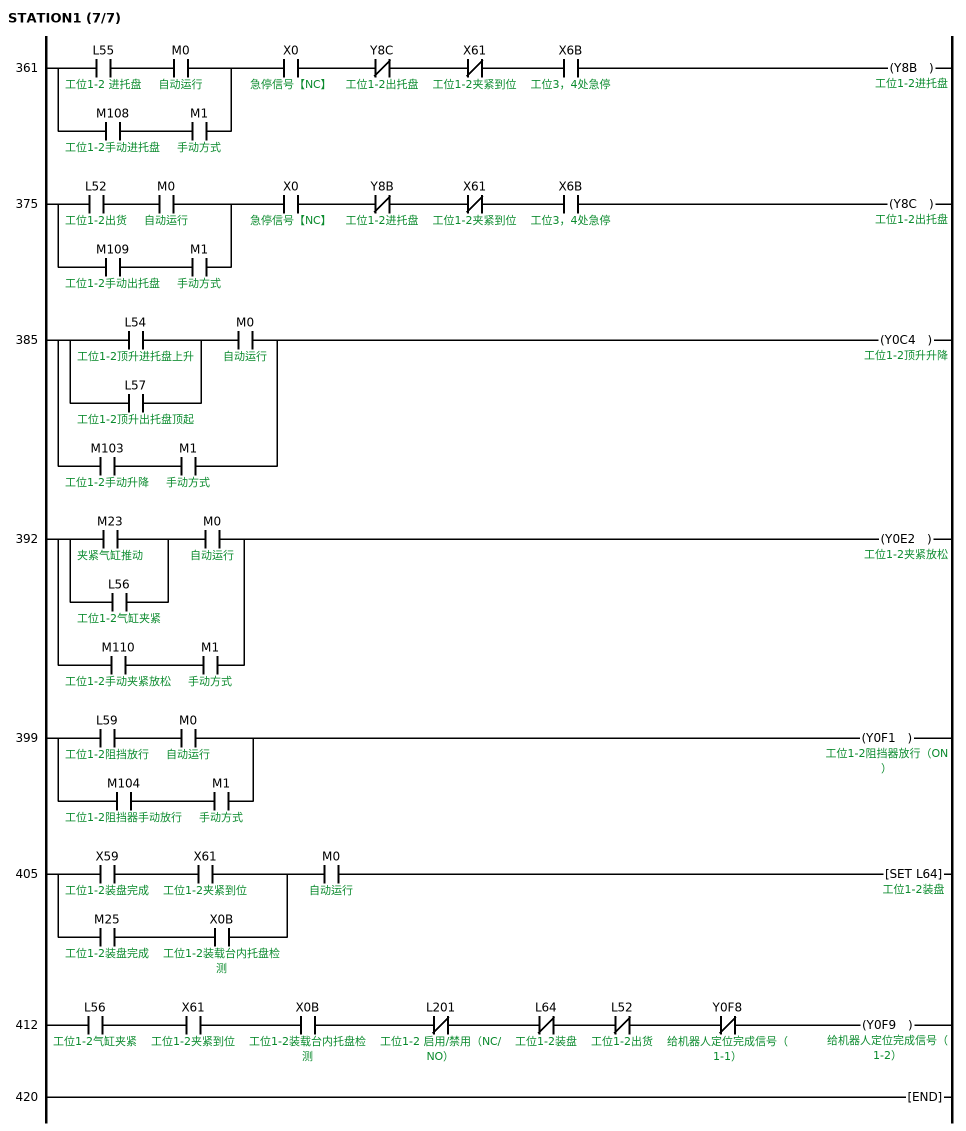
[picture p48: ladder of STATION1, rungs at steps 361 to 420]
361   LD      L55  ; 工位1-2 进托盘
      AND     M0  ; 自动运行
      LD      M108  ; 工位1-2手动进托盘
      AND     M1  ; 手动方式
      ORB
      AND     X0  ; 急停信号【NC】
      ANI     Y8C  ; 工位1-2出托盘
      ANI     X61  ; 工位1-2夹紧到位
      AND     X6B  ; 工位3，4处急停
      OUT     Y8B  ; 工位1-2进托盘
        [note] 1-2
375   LD      L52  ; 工位1-2出货
      AND     M0  ; 自动运行
      LD      M109  ; 工位1-2手动出托盘
      AND     M1  ; 手动方式
      ORB
      AND     X0  ; 急停信号【NC】
      ANI     Y8B  ; 工位1-2进托盘
      ANI     X61  ; 工位1-2夹紧到位
      AND     X6B  ; 工位3，4处急停
      OUT     Y8C  ; 工位1-2出托盘
385   LD      L54  ; 工位1-2顶升进托盘上升
      OR      L57  ; 工位1-2顶升出托盘顶起
      AND     M0  ; 自动运行
      LD      M103  ; 工位1-2手动升降
      AND     M1  ; 手动方式
      ORB
      OUT     Y0C4  ; 工位1-2顶升升降
392   LD      M23  ; 夹紧气缸推动
      OR      L56  ; 工位1-2气缸夹紧
      AND     M0  ; 自动运行
      LD      M110  ; 工位1-2手动夹紧放松
      AND     M1  ; 手动方式
      ORB
      OUT     Y0E2  ; 工位1-2夹紧放松
399   LD      L59  ; 工位1-2阻挡放行
      AND     M0  ; 自动运行
      LD      M104  ; 工位1-2阻挡器手动放行
      AND     M1  ; 手动方式
      ORB
      OUT     Y0F1  ; 工位1-2阻挡器放行（ON）
405   LD      X59  ; 工位1-2装盘完成
      AND     X61  ; 工位1-2夹紧到位
      LD      M25  ; 工位1-2装盘完成
      AND     X0B  ; 工位1-2装载台内托盘检测
      ORB
      AND     M0  ; 自动运行
      SET     L64  ; 工位1-2装盘
412   LD      L56  ; 工位1-2气缸夹紧
      AND     X61  ; 工位1-2夹紧到位
      AND     X0B  ; 工位1-2装载台内托盘检测
      ANI     L201  ; 工位1-2 启用/禁用（NC/NO）
      ANI     L64  ; 工位1-2装盘
      ANI     L52  ; 工位1-2出货
      ANI     Y0F8  ; 给机器人定位完成信号（1-1）
      OUT     Y0F9  ; 给机器人定位完成信号（1-2）
420   END
END_PROGRAM

PROGRAM STATION2
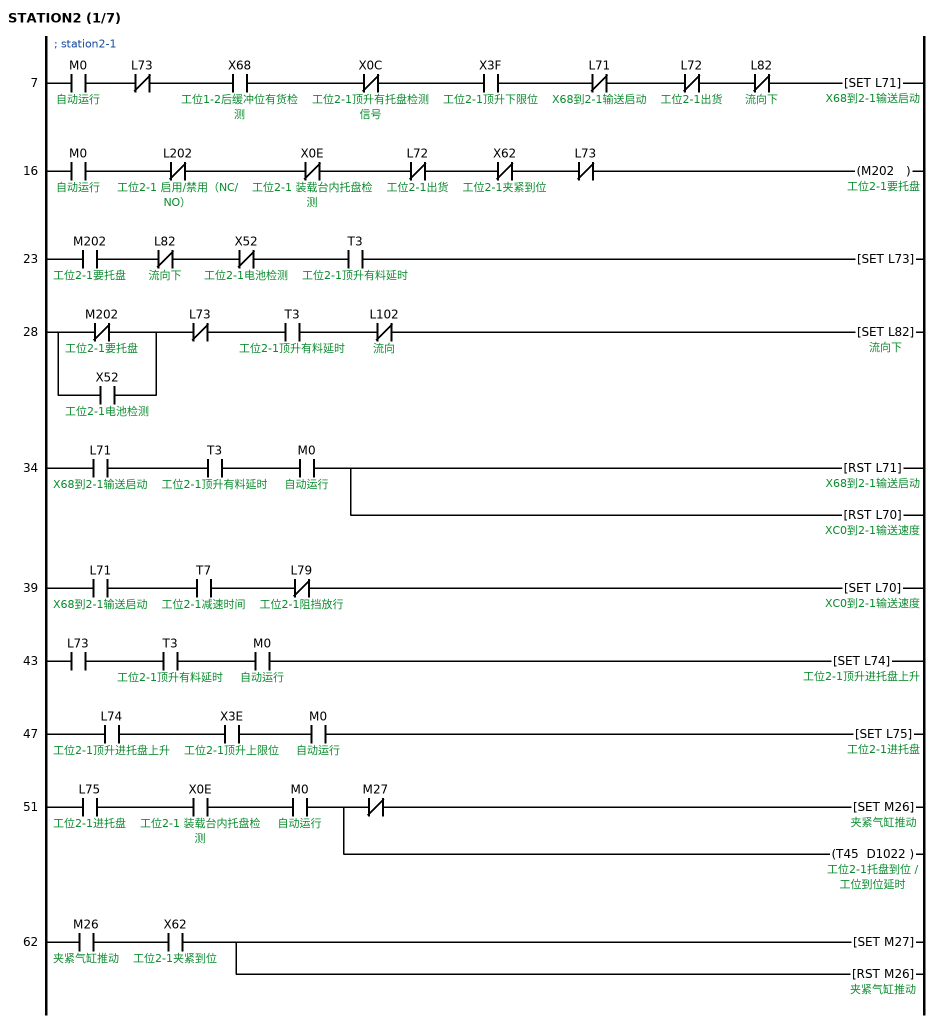
; station2-1
7     LD      M0  ; 自动运行
      ANI     L73
      AND     X68  ; 工位1-2后缓冲位有货检测
      ANI     X0C  ; 工位2-1顶升有托盘检测信号
      AND     X3F  ; 工位2-1顶升下限位
      ANI     L71  ; X68到2-1输送启动
      ANI     L72  ; 工位2-1出货
      ANI     L82  ; 流向下
      SET     L71  ; X68到2-1输送启动
16    LD      M0  ; 自动运行
      ANI     L202  ; 工位2-1 启用/禁用（NC/NO）
      ANI     X0E  ; 工位2-1 装载台内托盘检测
      ANI     L72  ; 工位2-1出货
      ANI     X62  ; 工位2-1夹紧到位
      ANI     L73
      OUT     M202  ; 工位2-1要托盘
23    LD      M202  ; 工位2-1要托盘
      ANI     L82  ; 流向下
      ANI     X52  ; 工位2-1电池检测
      AND     T3  ; 工位2-1顶升有料延时
      SET     L73
28    LDI     M202  ; 工位2-1要托盘
      OR      X52  ; 工位2-1电池检测
      ANI     L73
      AND     T3  ; 工位2-1顶升有料延时
      ANI     L102  ; 流向
      SET     L82  ; 流向下
34    LD      L71  ; X68到2-1输送启动
      AND     T3  ; 工位2-1顶升有料延时
      AND     M0  ; 自动运行
      RST     L71  ; X68到2-1输送启动
      RST     L70  ; XC0到2-1输送速度
39    LD      L71  ; X68到2-1输送启动
      AND     T7  ; 工位2-1减速时间
      ANI     L79  ; 工位2-1阻挡放行
      SET     L70  ; XC0到2-1输送速度
43    LD      L73
      AND     T3  ; 工位2-1顶升有料延时
      AND     M0  ; 自动运行
      SET     L74  ; 工位2-1顶升进托盘上升
47    LD      L74  ; 工位2-1顶升进托盘上升
      AND     X3E  ; 工位2-1顶升上限位
      AND     M0  ; 自动运行
      SET     L75  ; 工位2-1进托盘
51    LD      L75  ; 工位2-1进托盘
      AND     X0E  ; 工位2-1 装载台内托盘检测
      AND     M0  ; 自动运行
      MPS
      ANI     M27
      SET     M26  ; 夹紧气缸推动
      MPP
      OUT     T45 D1022  ; 工位2-1托盘到位 / 工位到位延时
62    LD      M26  ; 夹紧气缸推动
      AND     X62  ; 工位2-1夹紧到位
      SET     M27
      RST     M26  ; 夹紧气缸推动
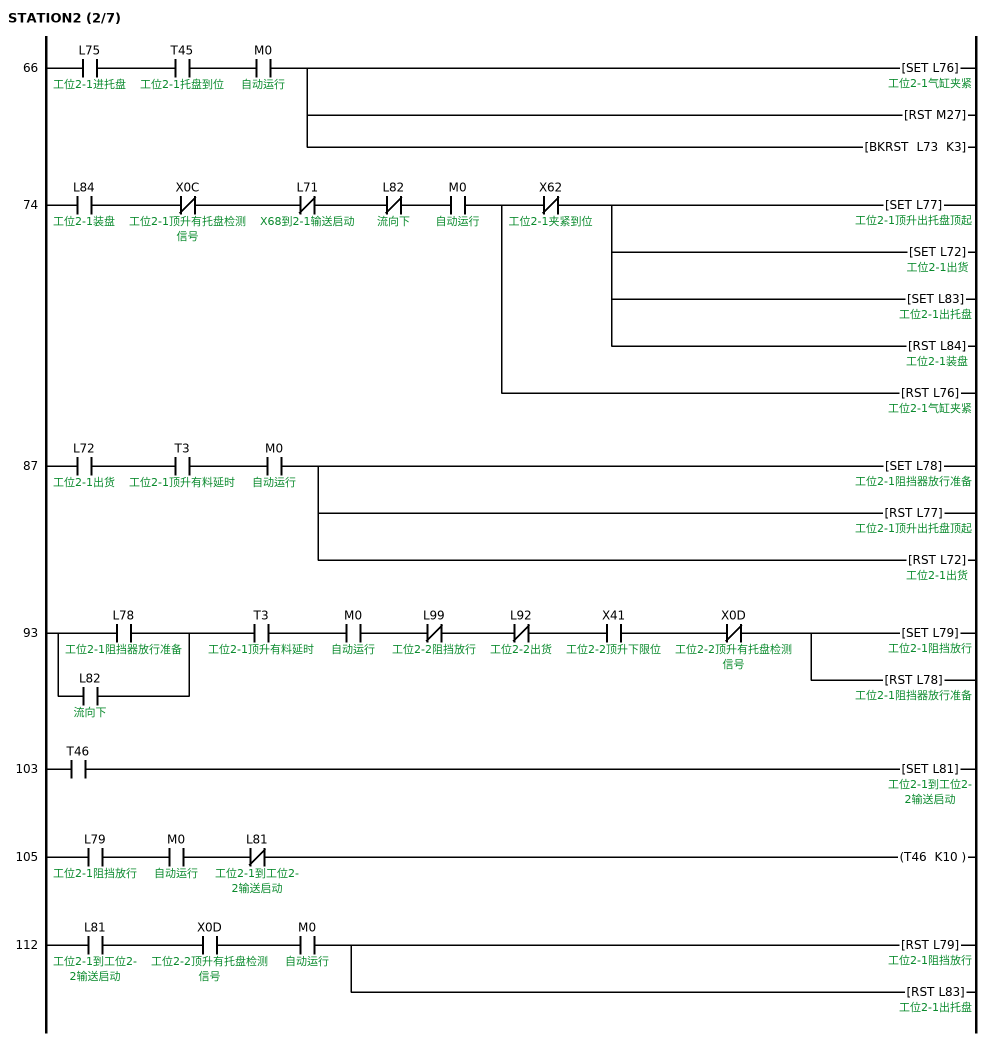
66    LD      L75  ; 工位2-1进托盘
      AND     T45  ; 工位2-1托盘到位
      AND     M0  ; 自动运行
      SET     L76  ; 工位2-1气缸夹紧
      RST     M27
      BKRST   L73 K3
74    LD      L84  ; 工位2-1装盘
      ANI     X0C  ; 工位2-1顶升有托盘检测信号
      ANI     L71  ; X68到2-1输送启动
      ANI     L82  ; 流向下
      AND     M0  ; 自动运行
      MPS
      ANI     X62  ; 工位2-1夹紧到位
      SET     L77  ; 工位2-1顶升出托盘顶起
      SET     L72  ; 工位2-1出货
      SET     L83  ; 工位2-1出托盘
      RST     L84  ; 工位2-1装盘
      MPP
      RST     L76  ; 工位2-1气缸夹紧
87    LD      L72  ; 工位2-1出货
      AND     T3  ; 工位2-1顶升有料延时
      AND     M0  ; 自动运行
      SET     L78  ; 工位2-1阻挡器放行准备
      RST     L77  ; 工位2-1顶升出托盘顶起
      RST     L72  ; 工位2-1出货
93    LD      L78  ; 工位2-1阻挡器放行准备
      OR      L82  ; 流向下
      AND     T3  ; 工位2-1顶升有料延时
      AND     M0  ; 自动运行
      ANI     L99  ; 工位2-2阻挡放行
      ANI     L92  ; 工位2-2出货
      AND     X41  ; 工位2-2顶升下限位
      ANI     X0D  ; 工位2-2顶升有托盘检测信号
      SET     L79  ; 工位2-1阻挡放行
      RST     L78  ; 工位2-1阻挡器放行准备
103   LD      T46
      SET     L81  ; 工位2-1到工位2-2输送启动
105   LD      L79  ; 工位2-1阻挡放行
      AND     M0  ; 自动运行
      ANI     L81  ; 工位2-1到工位2-2输送启动
      OUT     T46 K10
112   LD      L81  ; 工位2-1到工位2-2输送启动
      AND     X0D  ; 工位2-2顶升有托盘检测信号
      AND     M0  ; 自动运行
      RST     L79  ; 工位2-1阻挡放行
      RST     L83  ; 工位2-1出托盘
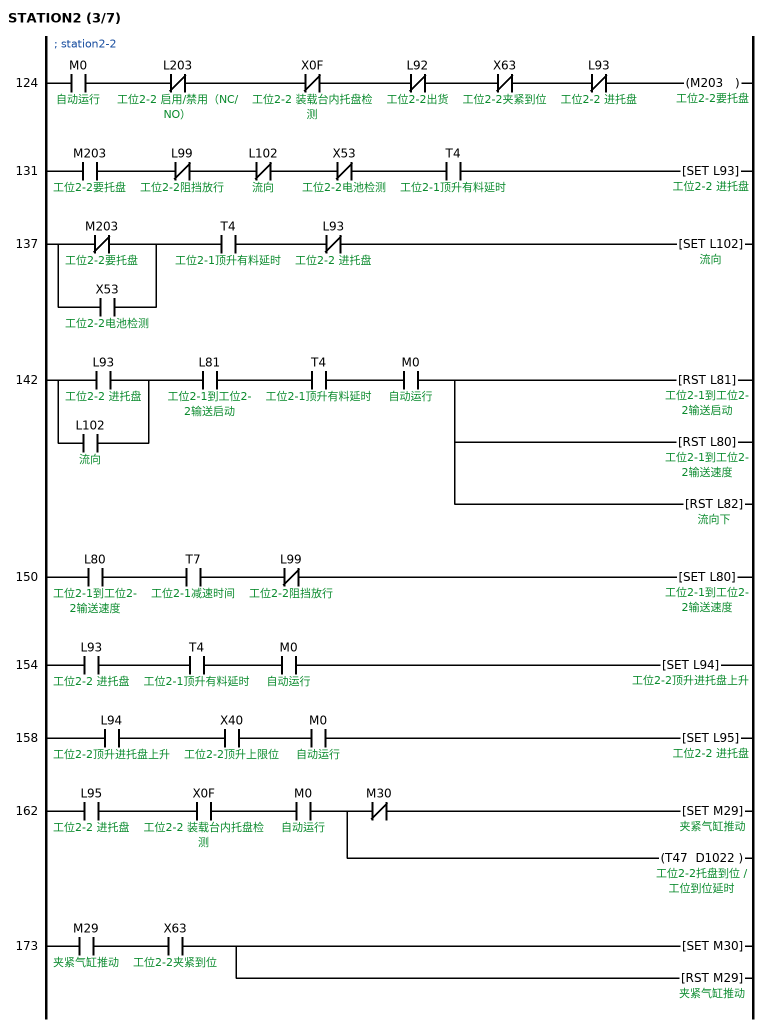
; station2-2
124   LD      M0  ; 自动运行
      ANI     L203  ; 工位2-2 启用/禁用（NC/NO）
      ANI     X0F  ; 工位2-2 装载台内托盘检测
      ANI     L92  ; 工位2-2出货
      ANI     X63  ; 工位2-2夹紧到位
      ANI     L93  ; 工位2-2 进托盘
      OUT     M203  ; 工位2-2要托盘
131   LD      M203  ; 工位2-2要托盘
      ANI     L99  ; 工位2-2阻挡放行
      ANI     L102  ; 流向
      ANI     X53  ; 工位2-2电池检测
      AND     T4  ; 工位2-1顶升有料延时
      SET     L93  ; 工位2-2 进托盘
137   LDI     M203  ; 工位2-2要托盘
      OR      X53  ; 工位2-2电池检测
      AND     T4  ; 工位2-1顶升有料延时
      ANI     L93  ; 工位2-2 进托盘
      SET     L102  ; 流向
142   LD      L93  ; 工位2-2 进托盘
      OR      L102  ; 流向
      AND     L81  ; 工位2-1到工位2-2输送启动
      AND     T4  ; 工位2-1顶升有料延时
      AND     M0  ; 自动运行
      RST     L81  ; 工位2-1到工位2-2输送启动
      RST     L80  ; 工位2-1到工位2-2输送速度
      RST     L82  ; 流向下
150   LD      L80  ; 工位2-1到工位2-2输送速度
      AND     T7  ; 工位2-1减速时间
      ANI     L99  ; 工位2-2阻挡放行
      SET     L80  ; 工位2-1到工位2-2输送速度
154   LD      L93  ; 工位2-2 进托盘
      AND     T4  ; 工位2-1顶升有料延时
      AND     M0  ; 自动运行
      SET     L94  ; 工位2-2顶升进托盘上升
158   LD      L94  ; 工位2-2顶升进托盘上升
      AND     X40  ; 工位2-2顶升上限位
      AND     M0  ; 自动运行
      SET     L95  ; 工位2-2 进托盘
162   LD      L95  ; 工位2-2 进托盘
      AND     X0F  ; 工位2-2 装载台内托盘检测
      AND     M0  ; 自动运行
      MPS
      ANI     M30
      SET     M29  ; 夹紧气缸推动
      MPP
      OUT     T47 D1022  ; 工位2-2托盘到位 / 工位到位延时
173   LD      M29  ; 夹紧气缸推动
      AND     X63  ; 工位2-2夹紧到位
      SET     M30
      RST     M29  ; 夹紧气缸推动
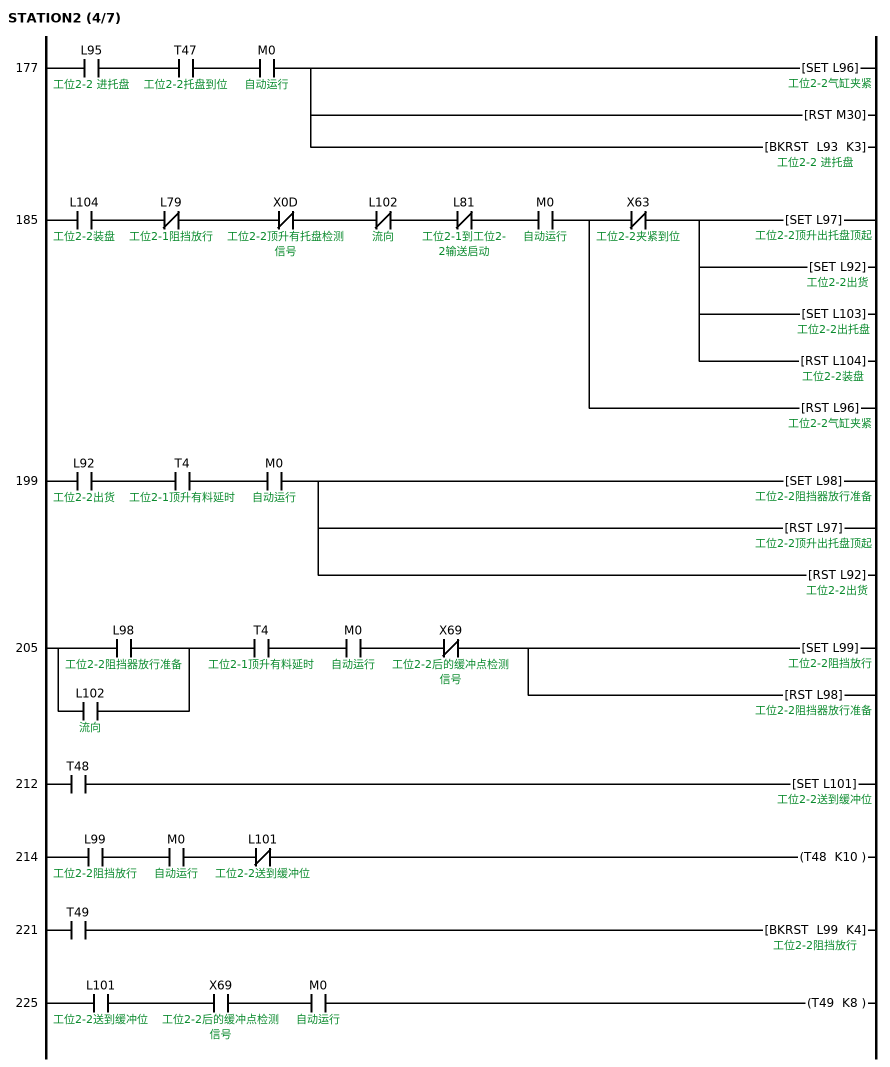
177   LD      L95  ; 工位2-2 进托盘
      AND     T47  ; 工位2-2托盘到位
      AND     M0  ; 自动运行
      SET     L96  ; 工位2-2气缸夹紧
      RST     M30
      BKRST   L93 K3
185   LD      L104  ; 工位2-2装盘
      ANI     L79  ; 工位2-1阻挡放行
      ANI     X0D  ; 工位2-2顶升有托盘检测信号
      ANI     L102  ; 流向
      ANI     L81  ; 工位2-1到工位2-2输送启动
      AND     M0  ; 自动运行
      MPS
      ANI     X63  ; 工位2-2夹紧到位
      SET     L97  ; 工位2-2顶升出托盘顶起
      SET     L92  ; 工位2-2出货
      SET     L103  ; 工位2-2出托盘
      RST     L104  ; 工位2-2装盘
      MPP
      RST     L96  ; 工位2-2气缸夹紧
199   LD      L92  ; 工位2-2出货
      AND     T4  ; 工位2-1顶升有料延时
      AND     M0  ; 自动运行
      SET     L98  ; 工位2-2阻挡器放行准备
      RST     L97  ; 工位2-2顶升出托盘顶起
      RST     L92  ; 工位2-2出货
205   LD      L98  ; 工位2-2阻挡器放行准备
      OR      L102  ; 流向
      AND     T4  ; 工位2-1顶升有料延时
      AND     M0  ; 自动运行
      ANI     X69  ; 工位2-2后的缓冲点检测信号
      SET     L99  ; 工位2-2阻挡放行
      RST     L98  ; 工位2-2阻挡器放行准备
212   LD      T48
      SET     L101  ; 工位2-2送到缓冲位
214   LD      L99  ; 工位2-2阻挡放行
      AND     M0  ; 自动运行
      ANI     L101  ; 工位2-2送到缓冲位
      OUT     T48 K10
221   LD      T49
      BKRST   L99 K4
225   LD      L101  ; 工位2-2送到缓冲位
      AND     X69  ; 工位2-2后的缓冲点检测信号
      AND     M0  ; 自动运行
      OUT     T49 K8
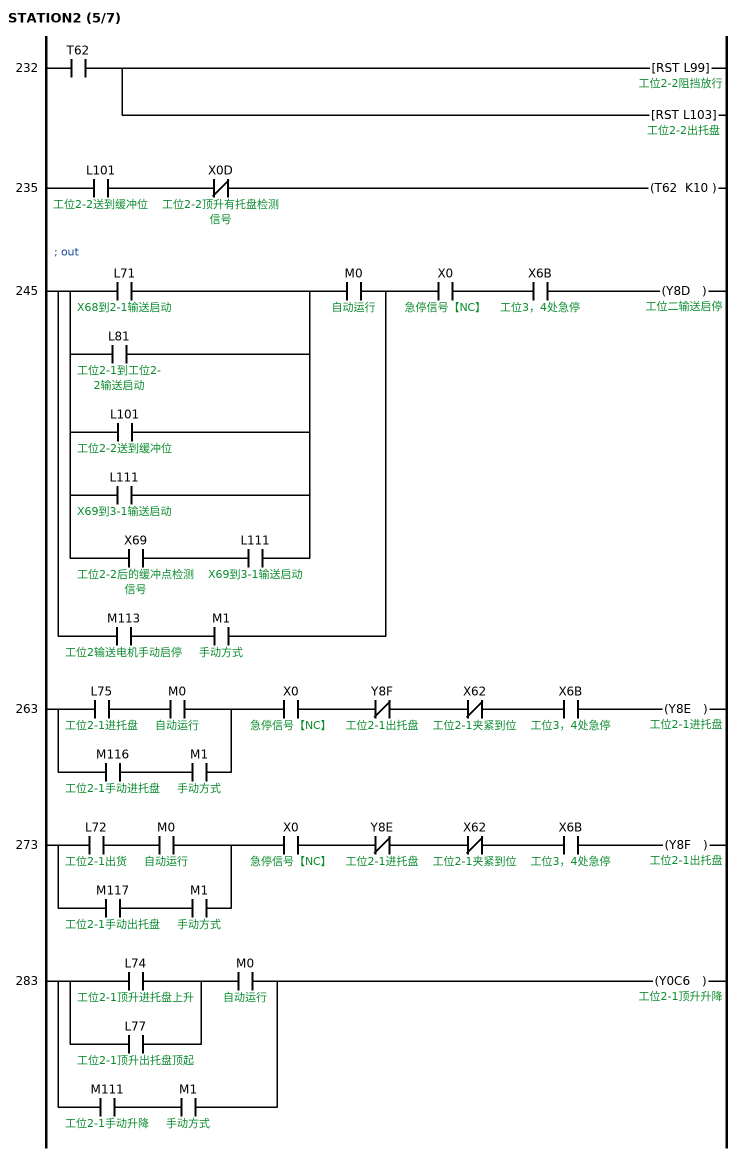
232   LD      T62
      RST     L99  ; 工位2-2阻挡放行
      RST     L103  ; 工位2-2出托盘
235   LD      L101  ; 工位2-2送到缓冲位
      ANI     X0D  ; 工位2-2顶升有托盘检测信号
      OUT     T62 K10
; out
245   LD      L71  ; X68到2-1输送启动
      OR      L81  ; 工位2-1到工位2-2输送启动
      OR      L101  ; 工位2-2送到缓冲位
      OR      L111  ; X69到3-1输送启动
      LD      X69  ; 工位2-2后的缓冲点检测信号
      AND     L111  ; X69到3-1输送启动
      ORB
      AND     M0  ; 自动运行
      LD      M113  ; 工位2输送电机手动启停
      AND     M1  ; 手动方式
      ORB
      AND     X0  ; 急停信号【NC】
      AND     X6B  ; 工位3，4处急停
      OUT     Y8D  ; 工位二输送启停
        [note] 1-1
263   LD      L75  ; 工位2-1进托盘
      AND     M0  ; 自动运行
      LD      M116  ; 工位2-1手动进托盘
      AND     M1  ; 手动方式
      ORB
      AND     X0  ; 急停信号【NC】
      ANI     Y8F  ; 工位2-1出托盘
      ANI     X62  ; 工位2-1夹紧到位
      AND     X6B  ; 工位3，4处急停
      OUT     Y8E  ; 工位2-1进托盘
273   LD      L72  ; 工位2-1出货
      AND     M0  ; 自动运行
      LD      M117  ; 工位2-1手动出托盘
      AND     M1  ; 手动方式
      ORB
      AND     X0  ; 急停信号【NC】
      ANI     Y8E  ; 工位2-1进托盘
      ANI     X62  ; 工位2-1夹紧到位
      AND     X6B  ; 工位3，4处急停
      OUT     Y8F  ; 工位2-1出托盘
283   LD      L74  ; 工位2-1顶升进托盘上升
      OR      L77  ; 工位2-1顶升出托盘顶起
      AND     M0  ; 自动运行
      LD      M111  ; 工位2-1手动升降
      AND     M1  ; 手动方式
      ORB
      OUT     Y0C6  ; 工位2-1顶升升降
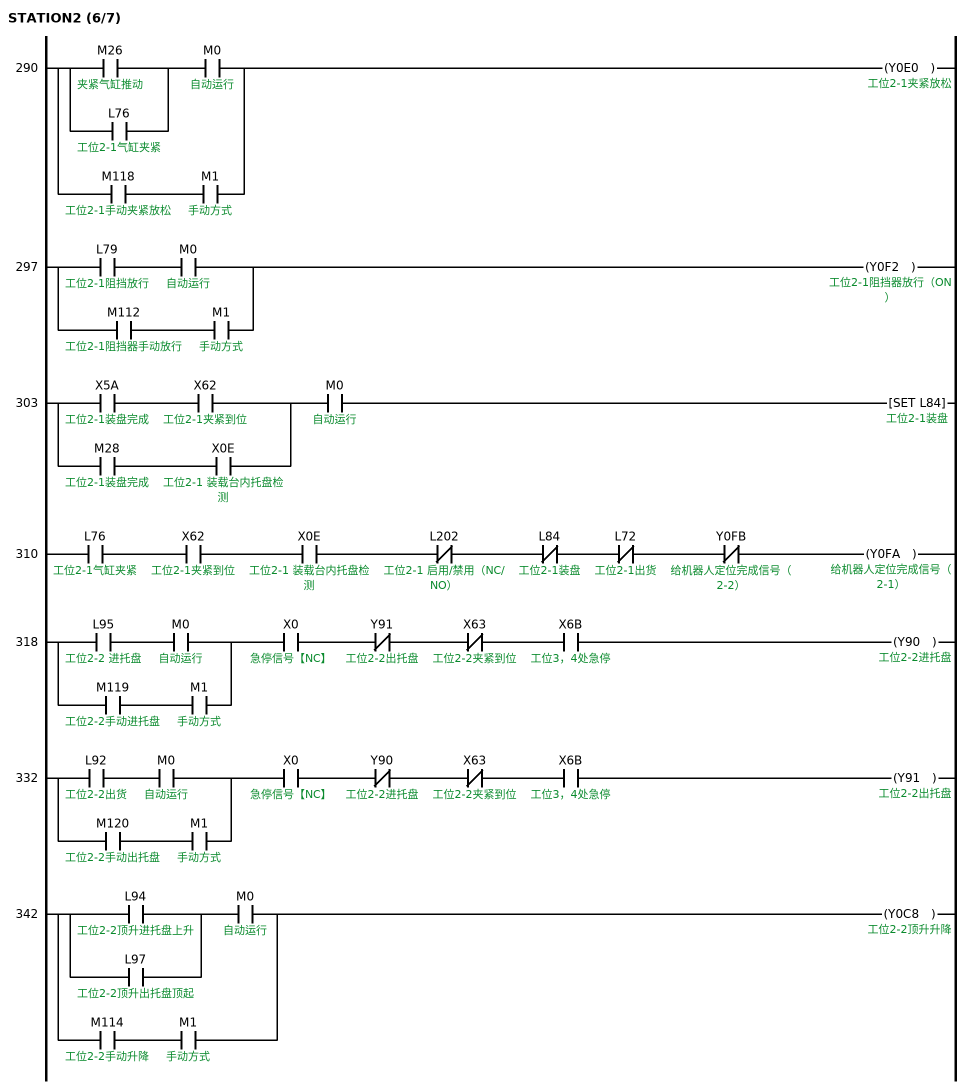
290   LD      M26  ; 夹紧气缸推动
      OR      L76  ; 工位2-1气缸夹紧
      AND     M0  ; 自动运行
      LD      M118  ; 工位2-1手动夹紧放松
      AND     M1  ; 手动方式
      ORB
      OUT     Y0E0  ; 工位2-1夹紧放松
297   LD      L79  ; 工位2-1阻挡放行
      AND     M0  ; 自动运行
      LD      M112  ; 工位2-1阻挡器手动放行
      AND     M1  ; 手动方式
      ORB
      OUT     Y0F2  ; 工位2-1阻挡器放行（ON）
303   LD      X5A  ; 工位2-1装盘完成
      AND     X62  ; 工位2-1夹紧到位
      LD      M28  ; 工位2-1装盘完成
      AND     X0E  ; 工位2-1 装载台内托盘检测
      ORB
      AND     M0  ; 自动运行
      SET     L84  ; 工位2-1装盘
310   LD      L76  ; 工位2-1气缸夹紧
      AND     X62  ; 工位2-1夹紧到位
      AND     X0E  ; 工位2-1 装载台内托盘检测
      ANI     L202  ; 工位2-1 启用/禁用（NC/NO）
      ANI     L84  ; 工位2-1装盘
      ANI     L72  ; 工位2-1出货
      ANI     Y0FB  ; 给机器人定位完成信号（2-2）
      OUT     Y0FA  ; 给机器人定位完成信号（2-1）
318   LD      L95  ; 工位2-2 进托盘
      AND     M0  ; 自动运行
      LD      M119  ; 工位2-2手动进托盘
      AND     M1  ; 手动方式
      ORB
      AND     X0  ; 急停信号【NC】
      ANI     Y91  ; 工位2-2出托盘
      ANI     X63  ; 工位2-2夹紧到位
      AND     X6B  ; 工位3，4处急停
      OUT     Y90  ; 工位2-2进托盘
        [note] 1-2
332   LD      L92  ; 工位2-2出货
      AND     M0  ; 自动运行
      LD      M120  ; 工位2-2手动出托盘
      AND     M1  ; 手动方式
      ORB
      AND     X0  ; 急停信号【NC】
      ANI     Y90  ; 工位2-2进托盘
      ANI     X63  ; 工位2-2夹紧到位
      AND     X6B  ; 工位3，4处急停
      OUT     Y91  ; 工位2-2出托盘
342   LD      L94  ; 工位2-2顶升进托盘上升
      OR      L97  ; 工位2-2顶升出托盘顶起
      AND     M0  ; 自动运行
      LD      M114  ; 工位2-2手动升降
      AND     M1  ; 手动方式
      ORB
      OUT     Y0C8  ; 工位2-2顶升升降
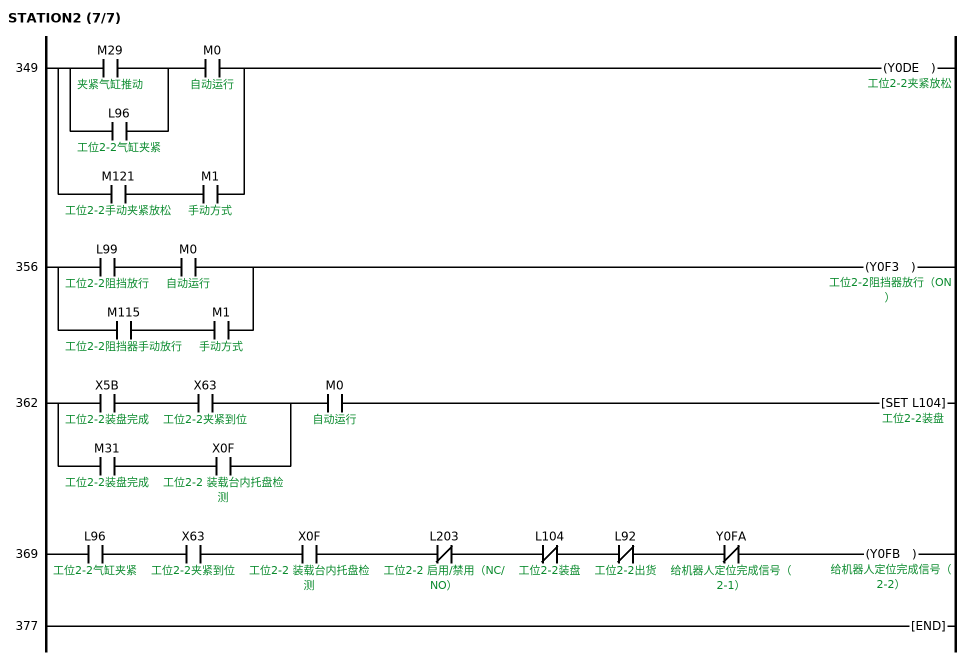
349   LD      M29  ; 夹紧气缸推动
      OR      L96  ; 工位2-2气缸夹紧
      AND     M0  ; 自动运行
      LD      M121  ; 工位2-2手动夹紧放松
      AND     M1  ; 手动方式
      ORB
      OUT     Y0DE  ; 工位2-2夹紧放松
356   LD      L99  ; 工位2-2阻挡放行
      AND     M0  ; 自动运行
      LD      M115  ; 工位2-2阻挡器手动放行
      AND     M1  ; 手动方式
      ORB
      OUT     Y0F3  ; 工位2-2阻挡器放行（ON）
362   LD      X5B  ; 工位2-2装盘完成
      AND     X63  ; 工位2-2夹紧到位
      LD      M31  ; 工位2-2装盘完成
      AND     X0F  ; 工位2-2 装载台内托盘检测
      ORB
      AND     M0  ; 自动运行
      SET     L104  ; 工位2-2装盘
369   LD      L96  ; 工位2-2气缸夹紧
      AND     X63  ; 工位2-2夹紧到位
      AND     X0F  ; 工位2-2 装载台内托盘检测
      ANI     L203  ; 工位2-2 启用/禁用（NC/NO）
      ANI     L104  ; 工位2-2装盘
      ANI     L92  ; 工位2-2出货
      ANI     Y0FA  ; 给机器人定位完成信号（2-1）
      OUT     Y0FB  ; 给机器人定位完成信号（2-2）
377   END
END_PROGRAM

PROGRAM STATION3
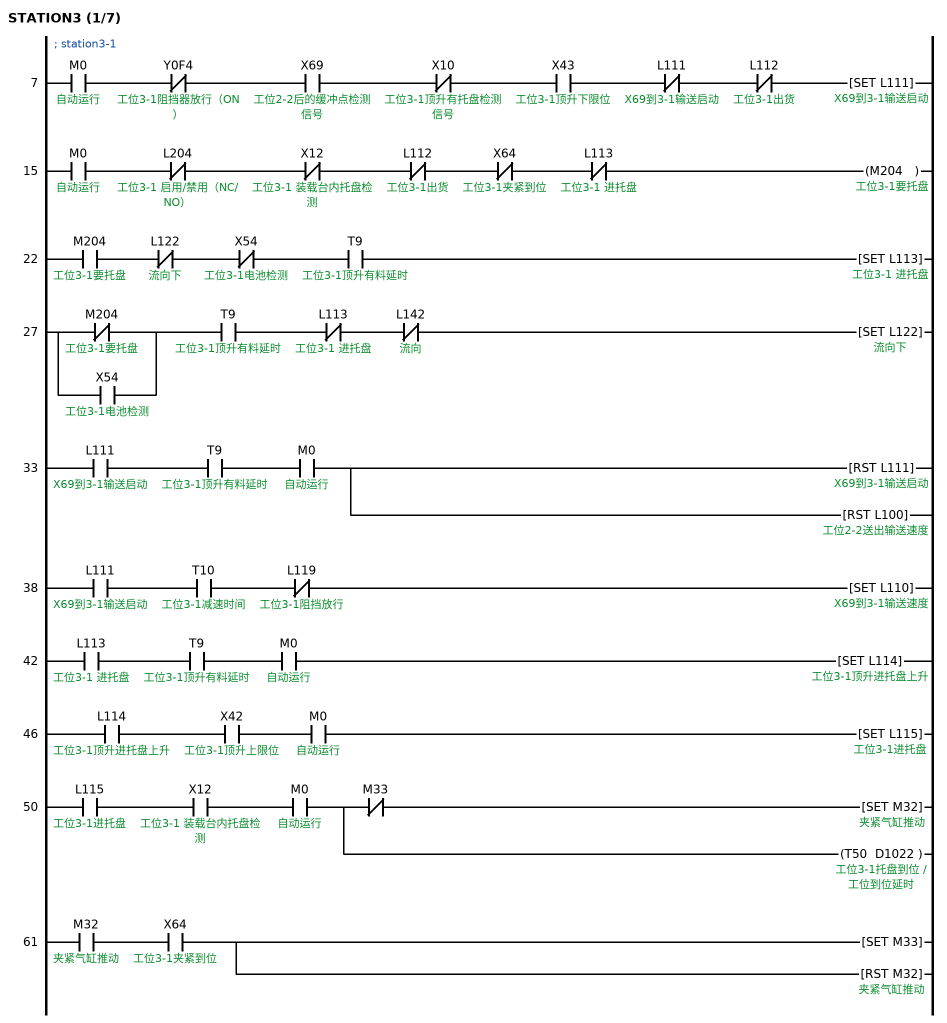
; station3-1
7     LD      M0  ; 自动运行
      ANI     Y0F4  ; 工位3-1阻挡器放行（ON）
      AND     X69  ; 工位2-2后的缓冲点检测信号
      ANI     X10  ; 工位3-1顶升有托盘检测信号
      AND     X43  ; 工位3-1顶升下限位
      ANI     L111  ; X69到3-1输送启动
      ANI     L112  ; 工位3-1出货
      SET     L111  ; X69到3-1输送启动
15    LD      M0  ; 自动运行
      ANI     L204  ; 工位3-1 启用/禁用（NC/NO）
      ANI     X12  ; 工位3-1 装载台内托盘检测
      ANI     L112  ; 工位3-1出货
      ANI     X64  ; 工位3-1夹紧到位
      ANI     L113  ; 工位3-1 进托盘
      OUT     M204  ; 工位3-1要托盘
22    LD      M204  ; 工位3-1要托盘
      ANI     L122  ; 流向下
      ANI     X54  ; 工位3-1电池检测
      AND     T9  ; 工位3-1顶升有料延时
      SET     L113  ; 工位3-1 进托盘
27    LDI     M204  ; 工位3-1要托盘
      OR      X54  ; 工位3-1电池检测
      AND     T9  ; 工位3-1顶升有料延时
      ANI     L113  ; 工位3-1 进托盘
      ANI     L142  ; 流向
      SET     L122  ; 流向下
33    LD      L111  ; X69到3-1输送启动
      AND     T9  ; 工位3-1顶升有料延时
      AND     M0  ; 自动运行
      RST     L111  ; X69到3-1输送启动
      RST     L100  ; 工位2-2送出输送速度
38    LD      L111  ; X69到3-1输送启动
      AND     T10  ; 工位3-1减速时间
      ANI     L119  ; 工位3-1阻挡放行
      SET     L110  ; X69到3-1输送速度
42    LD      L113  ; 工位3-1 进托盘
      AND     T9  ; 工位3-1顶升有料延时
      AND     M0  ; 自动运行
      SET     L114  ; 工位3-1顶升进托盘上升
46    LD      L114  ; 工位3-1顶升进托盘上升
      AND     X42  ; 工位3-1顶升上限位
      AND     M0  ; 自动运行
      SET     L115  ; 工位3-1进托盘
50    LD      L115  ; 工位3-1进托盘
      AND     X12  ; 工位3-1 装载台内托盘检测
      AND     M0  ; 自动运行
      MPS
      ANI     M33
      SET     M32  ; 夹紧气缸推动
      MPP
      OUT     T50 D1022  ; 工位3-1托盘到位 / 工位到位延时
61    LD      M32  ; 夹紧气缸推动
      AND     X64  ; 工位3-1夹紧到位
      SET     M33
      RST     M32  ; 夹紧气缸推动
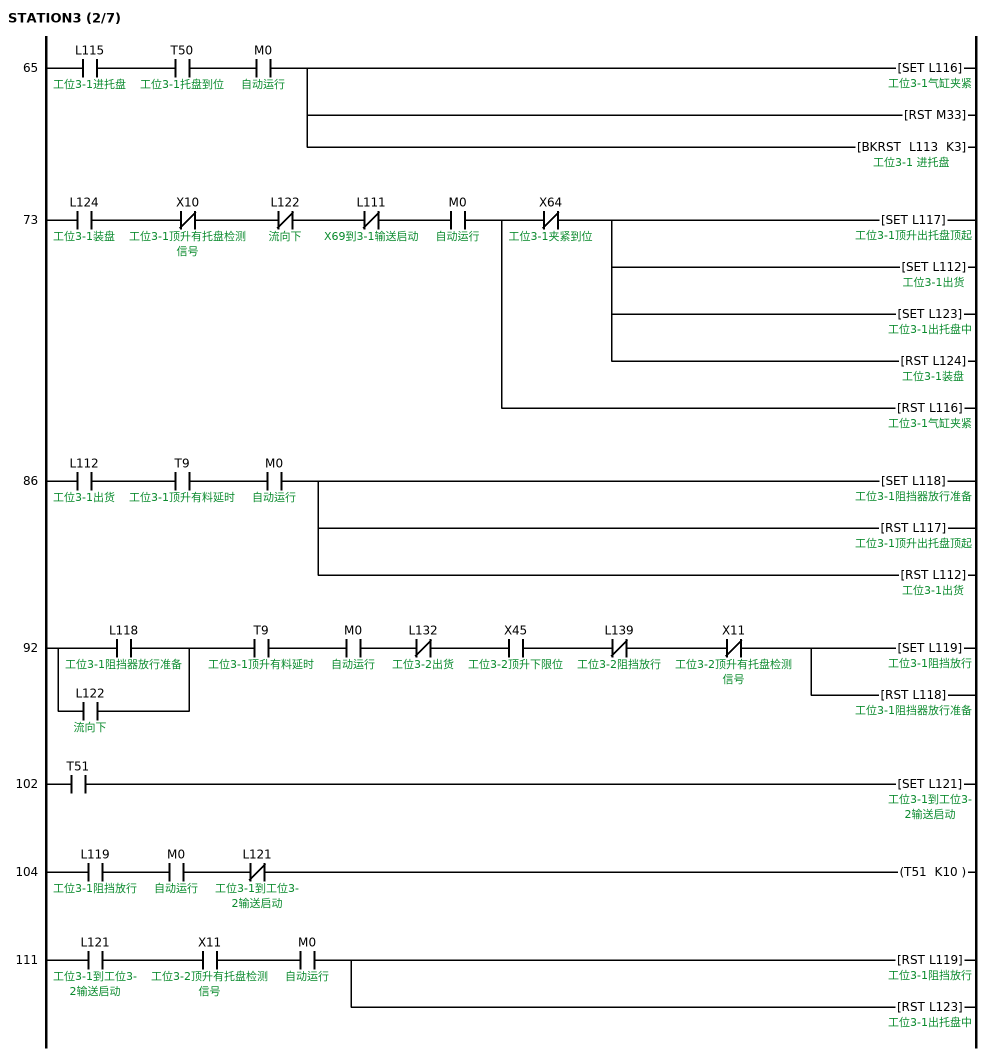
65    LD      L115  ; 工位3-1进托盘
      AND     T50  ; 工位3-1托盘到位
      AND     M0  ; 自动运行
      SET     L116  ; 工位3-1气缸夹紧
      RST     M33
      BKRST   L113 K3
73    LD      L124  ; 工位3-1装盘
      ANI     X10  ; 工位3-1顶升有托盘检测信号
      ANI     L122  ; 流向下
      ANI     L111  ; X69到3-1输送启动
      AND     M0  ; 自动运行
      MPS
      ANI     X64  ; 工位3-1夹紧到位
      SET     L117  ; 工位3-1顶升出托盘顶起
      SET     L112  ; 工位3-1出货
      SET     L123  ; 工位3-1出托盘中
      RST     L124  ; 工位3-1装盘
      MPP
      RST     L116  ; 工位3-1气缸夹紧
86    LD      L112  ; 工位3-1出货
      AND     T9  ; 工位3-1顶升有料延时
      AND     M0  ; 自动运行
      SET     L118  ; 工位3-1阻挡器放行准备
      RST     L117  ; 工位3-1顶升出托盘顶起
      RST     L112  ; 工位3-1出货
92    LD      L118  ; 工位3-1阻挡器放行准备
      OR      L122  ; 流向下
      AND     T9  ; 工位3-1顶升有料延时
      AND     M0  ; 自动运行
      ANI     L132  ; 工位3-2出货
      AND     X45  ; 工位3-2顶升下限位
      ANI     L139  ; 工位3-2阻挡放行
      ANI     X11  ; 工位3-2顶升有托盘检测信号
      SET     L119  ; 工位3-1阻挡放行
      RST     L118  ; 工位3-1阻挡器放行准备
102   LD      T51
      SET     L121  ; 工位3-1到工位3-2输送启动
104   LD      L119  ; 工位3-1阻挡放行
      AND     M0  ; 自动运行
      ANI     L121  ; 工位3-1到工位3-2输送启动
      OUT     T51 K10
111   LD      L121  ; 工位3-1到工位3-2输送启动
      AND     X11  ; 工位3-2顶升有托盘检测信号
      AND     M0  ; 自动运行
      RST     L119  ; 工位3-1阻挡放行
      RST     L123  ; 工位3-1出托盘中
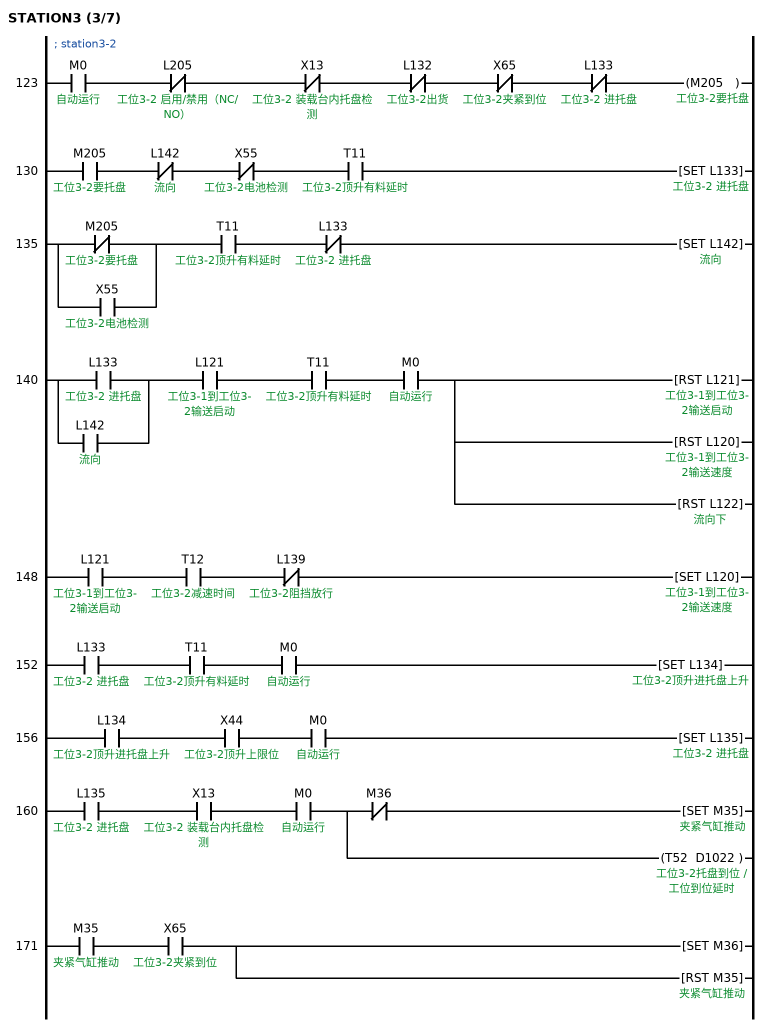
; station3-2
123   LD      M0  ; 自动运行
      ANI     L205  ; 工位3-2 启用/禁用（NC/NO）
      ANI     X13  ; 工位3-2 装载台内托盘检测
      ANI     L132  ; 工位3-2出货
      ANI     X65  ; 工位3-2夹紧到位
      ANI     L133  ; 工位3-2 进托盘
      OUT     M205  ; 工位3-2要托盘
130   LD      M205  ; 工位3-2要托盘
      ANI     L142  ; 流向
      ANI     X55  ; 工位3-2电池检测
      AND     T11  ; 工位3-2顶升有料延时
      SET     L133  ; 工位3-2 进托盘
135   LDI     M205  ; 工位3-2要托盘
      OR      X55  ; 工位3-2电池检测
      AND     T11  ; 工位3-2顶升有料延时
      ANI     L133  ; 工位3-2 进托盘
      SET     L142  ; 流向
140   LD      L133  ; 工位3-2 进托盘
      OR      L142  ; 流向
      AND     L121  ; 工位3-1到工位3-2输送启动
      AND     T11  ; 工位3-2顶升有料延时
      AND     M0  ; 自动运行
      RST     L121  ; 工位3-1到工位3-2输送启动
      RST     L120  ; 工位3-1到工位3-2输送速度
      RST     L122  ; 流向下
148   LD      L121  ; 工位3-1到工位3-2输送启动
      AND     T12  ; 工位3-2减速时间
      ANI     L139  ; 工位3-2阻挡放行
      SET     L120  ; 工位3-1到工位3-2输送速度
152   LD      L133  ; 工位3-2 进托盘
      AND     T11  ; 工位3-2顶升有料延时
      AND     M0  ; 自动运行
      SET     L134  ; 工位3-2顶升进托盘上升
156   LD      L134  ; 工位3-2顶升进托盘上升
      AND     X44  ; 工位3-2顶升上限位
      AND     M0  ; 自动运行
      SET     L135  ; 工位3-2 进托盘
160   LD      L135  ; 工位3-2 进托盘
      AND     X13  ; 工位3-2 装载台内托盘检测
      AND     M0  ; 自动运行
      MPS
      ANI     M36
      SET     M35  ; 夹紧气缸推动
      MPP
      OUT     T52 D1022  ; 工位3-2托盘到位 / 工位到位延时
171   LD      M35  ; 夹紧气缸推动
      AND     X65  ; 工位3-2夹紧到位
      SET     M36
      RST     M35  ; 夹紧气缸推动
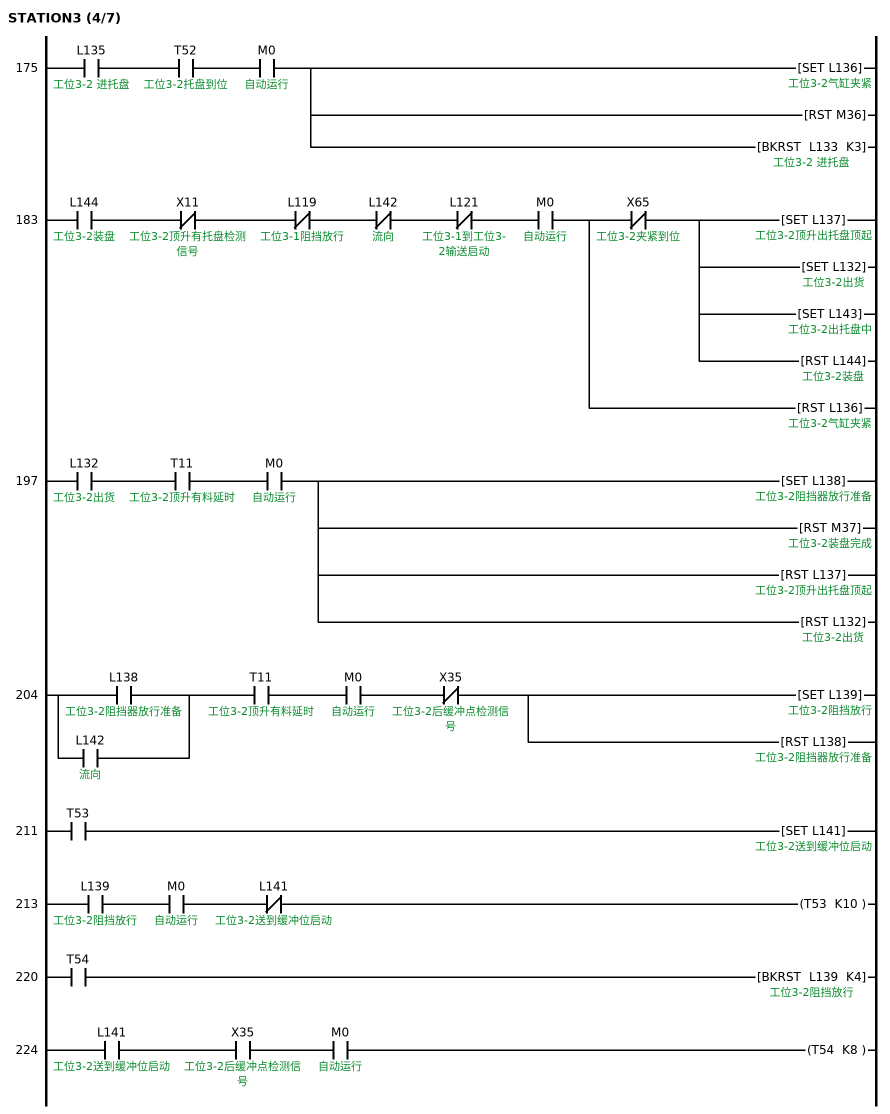
175   LD      L135  ; 工位3-2 进托盘
      AND     T52  ; 工位3-2托盘到位
      AND     M0  ; 自动运行
      SET     L136  ; 工位3-2气缸夹紧
      RST     M36
      BKRST   L133 K3
183   LD      L144  ; 工位3-2装盘
      ANI     X11  ; 工位3-2顶升有托盘检测信号
      ANI     L119  ; 工位3-1阻挡放行
      ANI     L142  ; 流向
      ANI     L121  ; 工位3-1到工位3-2输送启动
      AND     M0  ; 自动运行
      MPS
      ANI     X65  ; 工位3-2夹紧到位
      SET     L137  ; 工位3-2顶升出托盘顶起
      SET     L132  ; 工位3-2出货
      SET     L143  ; 工位3-2出托盘中
      RST     L144  ; 工位3-2装盘
      MPP
      RST     L136  ; 工位3-2气缸夹紧
197   LD      L132  ; 工位3-2出货
      AND     T11  ; 工位3-2顶升有料延时
      AND     M0  ; 自动运行
      SET     L138  ; 工位3-2阻挡器放行准备
      RST     M37  ; 工位3-2装盘完成
      RST     L137  ; 工位3-2顶升出托盘顶起
      RST     L132  ; 工位3-2出货
204   LD      L138  ; 工位3-2阻挡器放行准备
      OR      L142  ; 流向
      AND     T11  ; 工位3-2顶升有料延时
      AND     M0  ; 自动运行
      ANI     X35  ; 工位3-2后缓冲点检测信号
      SET     L139  ; 工位3-2阻挡放行
      RST     L138  ; 工位3-2阻挡器放行准备
211   LD      T53
      SET     L141  ; 工位3-2送到缓冲位启动
213   LD      L139  ; 工位3-2阻挡放行
      AND     M0  ; 自动运行
      ANI     L141  ; 工位3-2送到缓冲位启动
      OUT     T53 K10
220   LD      T54
      BKRST   L139 K4
224   LD      L141  ; 工位3-2送到缓冲位启动
      AND     X35  ; 工位3-2后缓冲点检测信号
      AND     M0  ; 自动运行
      OUT     T54 K8
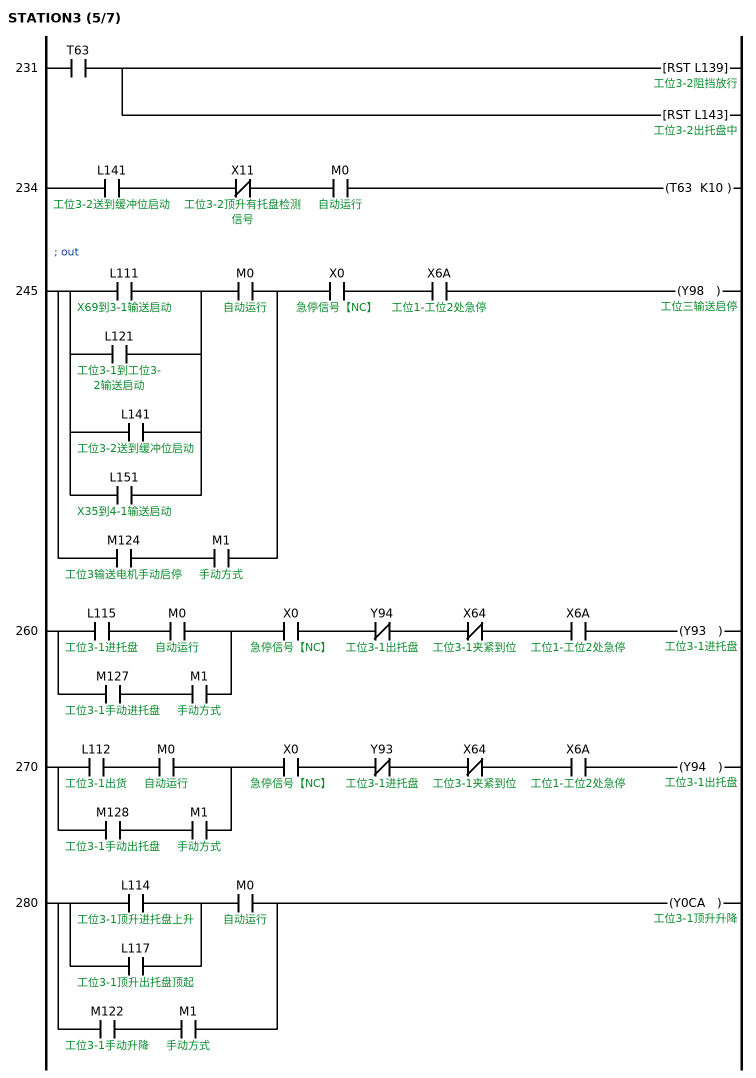
231   LD      T63
      RST     L139  ; 工位3-2阻挡放行
      RST     L143  ; 工位3-2出托盘中
234   LD      L141  ; 工位3-2送到缓冲位启动
      ANI     X11  ; 工位3-2顶升有托盘检测信号
      AND     M0  ; 自动运行
      OUT     T63 K10
; out
245   LD      L111  ; X69到3-1输送启动
      OR      L121  ; 工位3-1到工位3-2输送启动
      OR      L141  ; 工位3-2送到缓冲位启动
      OR      L151  ; X35到4-1输送启动
      AND     M0  ; 自动运行
      LD      M124  ; 工位3输送电机手动启停
      AND     M1  ; 手动方式
      ORB
      AND     X0  ; 急停信号【NC】
      AND     X6A  ; 工位1-工位2处急停
      OUT     Y98  ; 工位三输送启停
        [note] 3-1
260   LD      L115  ; 工位3-1进托盘
      AND     M0  ; 自动运行
      LD      M127  ; 工位3-1手动进托盘
      AND     M1  ; 手动方式
      ORB
      AND     X0  ; 急停信号【NC】
      ANI     Y94  ; 工位3-1出托盘
      ANI     X64  ; 工位3-1夹紧到位
      AND     X6A  ; 工位1-工位2处急停
      OUT     Y93  ; 工位3-1进托盘
270   LD      L112  ; 工位3-1出货
      AND     M0  ; 自动运行
      LD      M128  ; 工位3-1手动出托盘
      AND     M1  ; 手动方式
      ORB
      AND     X0  ; 急停信号【NC】
      ANI     Y93  ; 工位3-1进托盘
      ANI     X64  ; 工位3-1夹紧到位
      AND     X6A  ; 工位1-工位2处急停
      OUT     Y94  ; 工位3-1出托盘
280   LD      L114  ; 工位3-1顶升进托盘上升
      OR      L117  ; 工位3-1顶升出托盘顶起
      AND     M0  ; 自动运行
      LD      M122  ; 工位3-1手动升降
      AND     M1  ; 手动方式
      ORB
      OUT     Y0CA  ; 工位3-1顶升升降
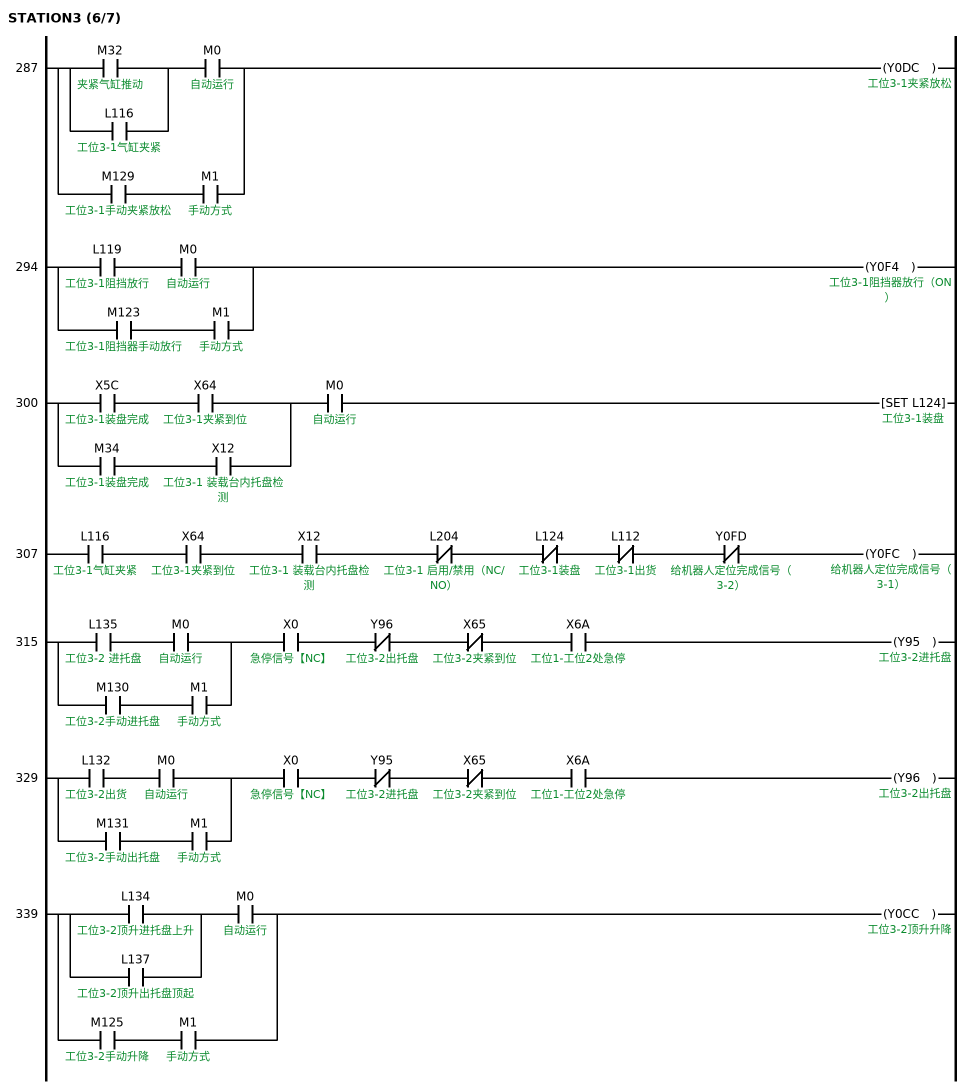
287   LD      M32  ; 夹紧气缸推动
      OR      L116  ; 工位3-1气缸夹紧
      AND     M0  ; 自动运行
      LD      M129  ; 工位3-1手动夹紧放松
      AND     M1  ; 手动方式
      ORB
      OUT     Y0DC  ; 工位3-1夹紧放松
294   LD      L119  ; 工位3-1阻挡放行
      AND     M0  ; 自动运行
      LD      M123  ; 工位3-1阻挡器手动放行
      AND     M1  ; 手动方式
      ORB
      OUT     Y0F4  ; 工位3-1阻挡器放行（ON）
300   LD      X5C  ; 工位3-1装盘完成
      AND     X64  ; 工位3-1夹紧到位
      LD      M34  ; 工位3-1装盘完成
      AND     X12  ; 工位3-1 装载台内托盘检测
      ORB
      AND     M0  ; 自动运行
      SET     L124  ; 工位3-1装盘
307   LD      L116  ; 工位3-1气缸夹紧
      AND     X64  ; 工位3-1夹紧到位
      AND     X12  ; 工位3-1 装载台内托盘检测
      ANI     L204  ; 工位3-1 启用/禁用（NC/NO）
      ANI     L124  ; 工位3-1装盘
      ANI     L112  ; 工位3-1出货
      ANI     Y0FD  ; 给机器人定位完成信号（3-2）
      OUT     Y0FC  ; 给机器人定位完成信号（3-1）
315   LD      L135  ; 工位3-2 进托盘
      AND     M0  ; 自动运行
      LD      M130  ; 工位3-2手动进托盘
      AND     M1  ; 手动方式
      ORB
      AND     X0  ; 急停信号【NC】
      ANI     Y96  ; 工位3-2出托盘
      ANI     X65  ; 工位3-2夹紧到位
      AND     X6A  ; 工位1-工位2处急停
      OUT     Y95  ; 工位3-2进托盘
        [note] 3-2
329   LD      L132  ; 工位3-2出货
      AND     M0  ; 自动运行
      LD      M131  ; 工位3-2手动出托盘
      AND     M1  ; 手动方式
      ORB
      AND     X0  ; 急停信号【NC】
      ANI     Y95  ; 工位3-2进托盘
      ANI     X65  ; 工位3-2夹紧到位
      AND     X6A  ; 工位1-工位2处急停
      OUT     Y96  ; 工位3-2出托盘
339   LD      L134  ; 工位3-2顶升进托盘上升
      OR      L137  ; 工位3-2顶升出托盘顶起
      AND     M0  ; 自动运行
      LD      M125  ; 工位3-2手动升降
      AND     M1  ; 手动方式
      ORB
      OUT     Y0CC  ; 工位3-2顶升升降
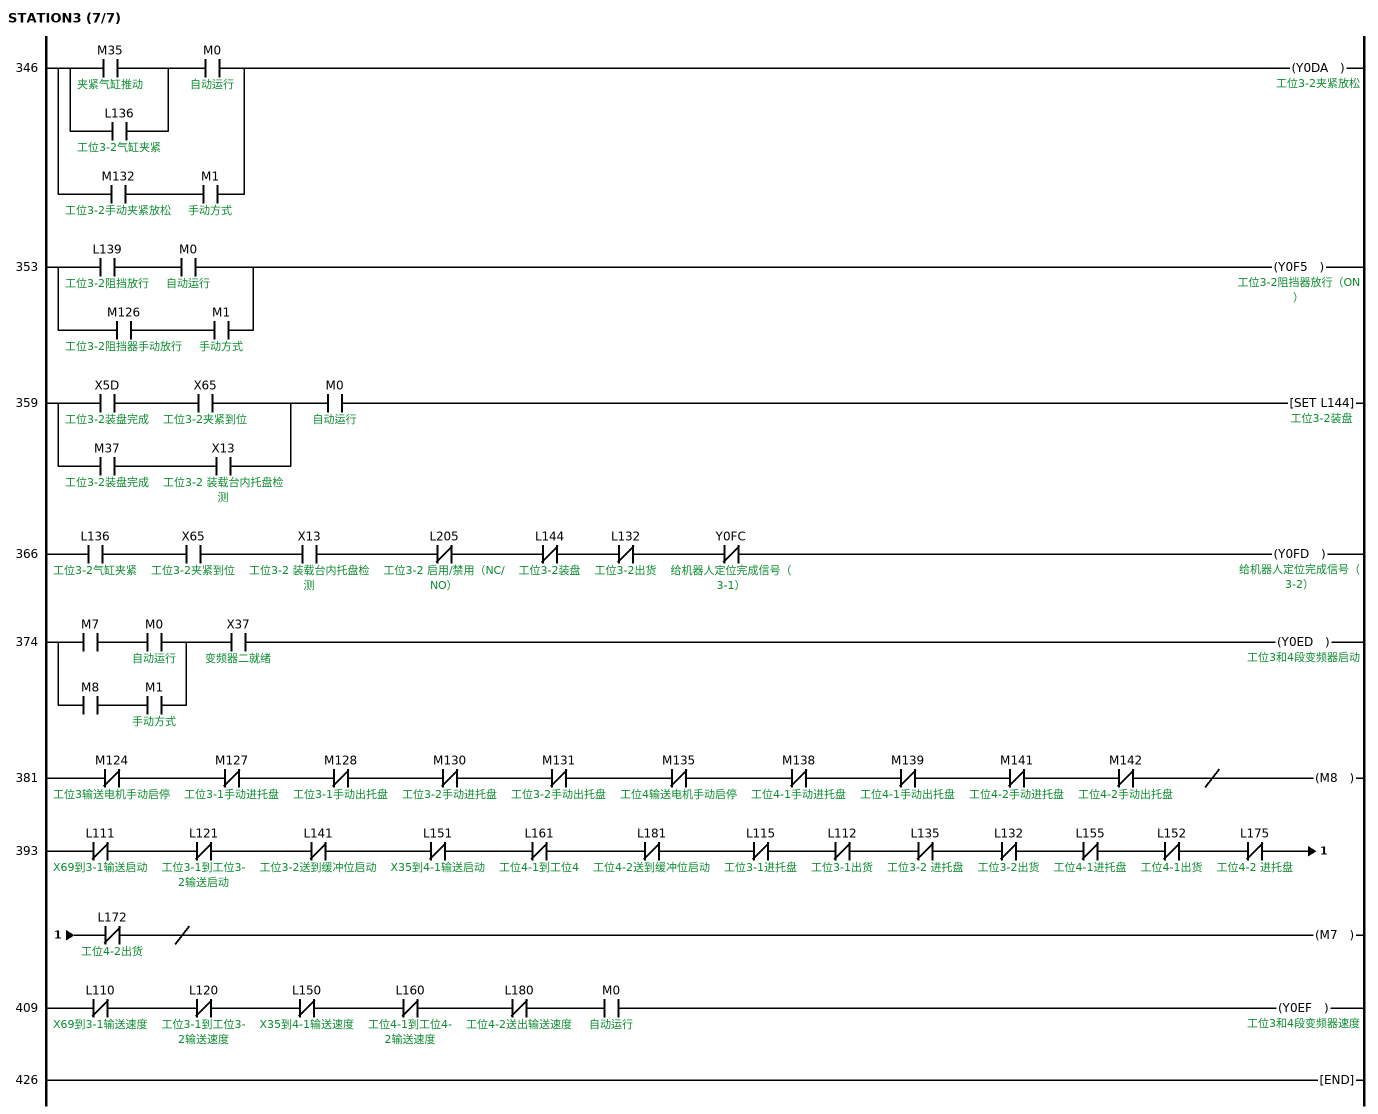
346   LD      M35  ; 夹紧气缸推动
      OR      L136  ; 工位3-2气缸夹紧
      AND     M0  ; 自动运行
      LD      M132  ; 工位3-2手动夹紧放松
      AND     M1  ; 手动方式
      ORB
      OUT     Y0DA  ; 工位3-2夹紧放松
353   LD      L139  ; 工位3-2阻挡放行
      AND     M0  ; 自动运行
      LD      M126  ; 工位3-2阻挡器手动放行
      AND     M1  ; 手动方式
      ORB
      OUT     Y0F5  ; 工位3-2阻挡器放行（ON）
359   LD      X5D  ; 工位3-2装盘完成
      AND     X65  ; 工位3-2夹紧到位
      LD      M37  ; 工位3-2装盘完成
      AND     X13  ; 工位3-2 装载台内托盘检测
      ORB
      AND     M0  ; 自动运行
      SET     L144  ; 工位3-2装盘
366   LD      L136  ; 工位3-2气缸夹紧
      AND     X65  ; 工位3-2夹紧到位
      AND     X13  ; 工位3-2 装载台内托盘检测
      ANI     L205  ; 工位3-2 启用/禁用（NC/NO）
      ANI     L144  ; 工位3-2装盘
      ANI     L132  ; 工位3-2出货
      ANI     Y0FC  ; 给机器人定位完成信号（3-1）
      OUT     Y0FD  ; 给机器人定位完成信号（3-2）
374   LD      M7
      AND     M0  ; 自动运行
      LD      M8
      AND     M1  ; 手动方式
      ORB
      AND     X37  ; 变频器二就绪
      OUT     Y0ED  ; 工位3和4段变频器启动
381   LDI     M124  ; 工位3输送电机手动启停
      ANI     M127  ; 工位3-1手动进托盘
      ANI     M128  ; 工位3-1手动出托盘
      ANI     M130  ; 工位3-2手动进托盘
      ANI     M131  ; 工位3-2手动出托盘
      ANI     M135  ; 工位4输送电机手动启停
      ANI     M138  ; 工位4-1手动进托盘
      ANI     M139  ; 工位4-1手动出托盘
      ANI     M141  ; 工位4-2手动进托盘
      ANI     M142  ; 工位4-2手动出托盘
      INV
      OUT     M8
393   LDI     L111  ; X69到3-1输送启动
      ANI     L121  ; 工位3-1到工位3-2输送启动
      ANI     L141  ; 工位3-2送到缓冲位启动
      ANI     L151  ; X35到4-1输送启动
      ANI     L161  ; 工位4-1到工位4
      ANI     L181  ; 工位4-2送到缓冲位启动
      ANI     L115  ; 工位3-1进托盘
      ANI     L112  ; 工位3-1出货
      ANI     L135  ; 工位3-2 进托盘
      ANI     L132  ; 工位3-2出货
      ANI     L155  ; 工位4-1进托盘
      ANI     L152  ; 工位4-1出货
      ANI     L175  ; 工位4-2 进托盘
      ANI     L172  ; 工位4-2出货
      INV
      OUT     M7
409   LDI     L110  ; X69到3-1输送速度
      ANI     L120  ; 工位3-1到工位3-2输送速度
      ANI     L150  ; X35到4-1输送速度
      ANI     L160  ; 工位4-1到工位4-2输送速度
      ANI     L180  ; 工位4-2送出输送速度
      AND     M0  ; 自动运行
      OUT     Y0EF  ; 工位3和4段变频器速度
        [note] ON高速，OFF低速
426   END
END_PROGRAM

PROGRAM STATION4
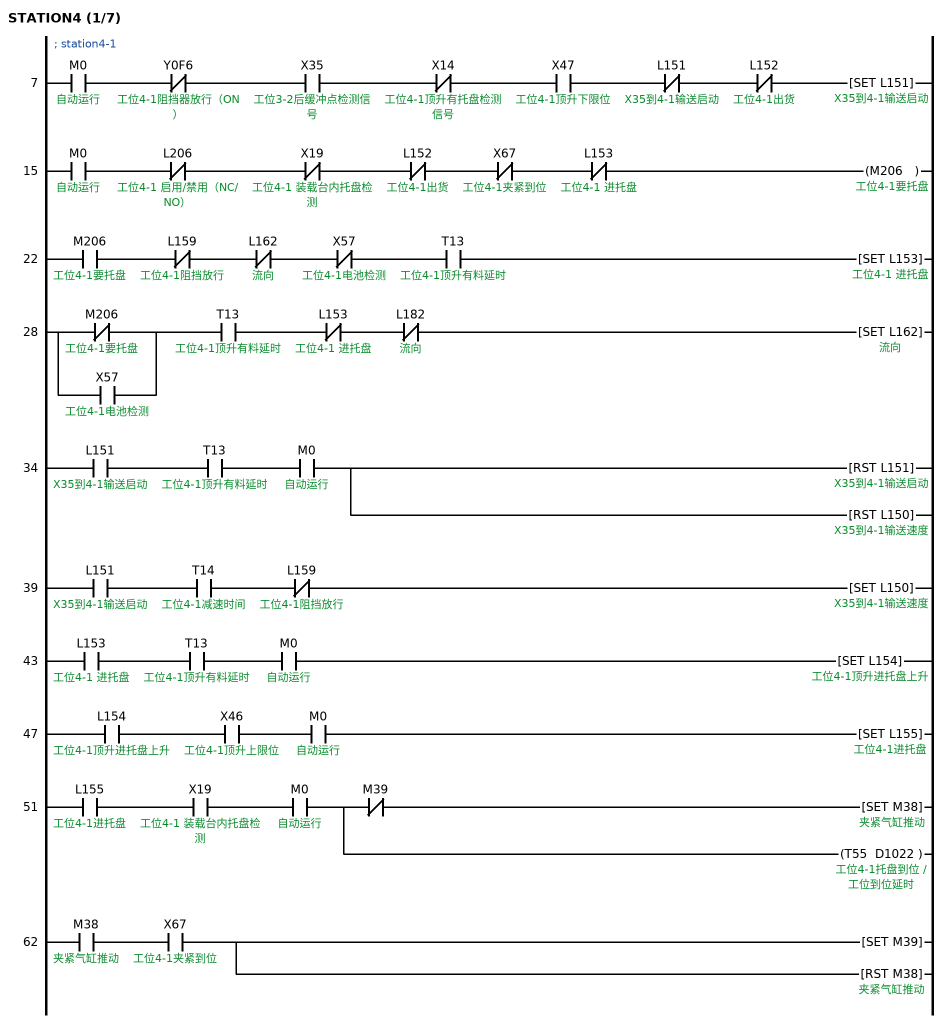
; station4-1
7     LD      M0  ; 自动运行
      ANI     Y0F6  ; 工位4-1阻挡器放行（ON）
      AND     X35  ; 工位3-2后缓冲点检测信号
      ANI     X14  ; 工位4-1顶升有托盘检测信号
      AND     X47  ; 工位4-1顶升下限位
      ANI     L151  ; X35到4-1输送启动
      ANI     L152  ; 工位4-1出货
      SET     L151  ; X35到4-1输送启动
15    LD      M0  ; 自动运行
      ANI     L206  ; 工位4-1 启用/禁用（NC/NO）
      ANI     X19  ; 工位4-1 装载台内托盘检测
      ANI     L152  ; 工位4-1出货
      ANI     X67  ; 工位4-1夹紧到位
      ANI     L153  ; 工位4-1 进托盘
      OUT     M206  ; 工位4-1要托盘
22    LD      M206  ; 工位4-1要托盘
      ANI     L159  ; 工位4-1阻挡放行
      ANI     L162  ; 流向
      ANI     X57  ; 工位4-1电池检测
      AND     T13  ; 工位4-1顶升有料延时
      SET     L153  ; 工位4-1 进托盘
28    LDI     M206  ; 工位4-1要托盘
      OR      X57  ; 工位4-1电池检测
      AND     T13  ; 工位4-1顶升有料延时
      ANI     L153  ; 工位4-1 进托盘
      ANI     L182  ; 流向
      SET     L162  ; 流向
34    LD      L151  ; X35到4-1输送启动
      AND     T13  ; 工位4-1顶升有料延时
      AND     M0  ; 自动运行
      RST     L151  ; X35到4-1输送启动
      RST     L150  ; X35到4-1输送速度
39    LD      L151  ; X35到4-1输送启动
      AND     T14  ; 工位4-1减速时间
      ANI     L159  ; 工位4-1阻挡放行
      SET     L150  ; X35到4-1输送速度
43    LD      L153  ; 工位4-1 进托盘
      AND     T13  ; 工位4-1顶升有料延时
      AND     M0  ; 自动运行
      SET     L154  ; 工位4-1顶升进托盘上升
47    LD      L154  ; 工位4-1顶升进托盘上升
      AND     X46  ; 工位4-1顶升上限位
      AND     M0  ; 自动运行
      SET     L155  ; 工位4-1进托盘
51    LD      L155  ; 工位4-1进托盘
      AND     X19  ; 工位4-1 装载台内托盘检测
      AND     M0  ; 自动运行
      MPS
      ANI     M39
      SET     M38  ; 夹紧气缸推动
      MPP
      OUT     T55 D1022  ; 工位4-1托盘到位 / 工位到位延时
62    LD      M38  ; 夹紧气缸推动
      AND     X67  ; 工位4-1夹紧到位
      SET     M39
      RST     M38  ; 夹紧气缸推动
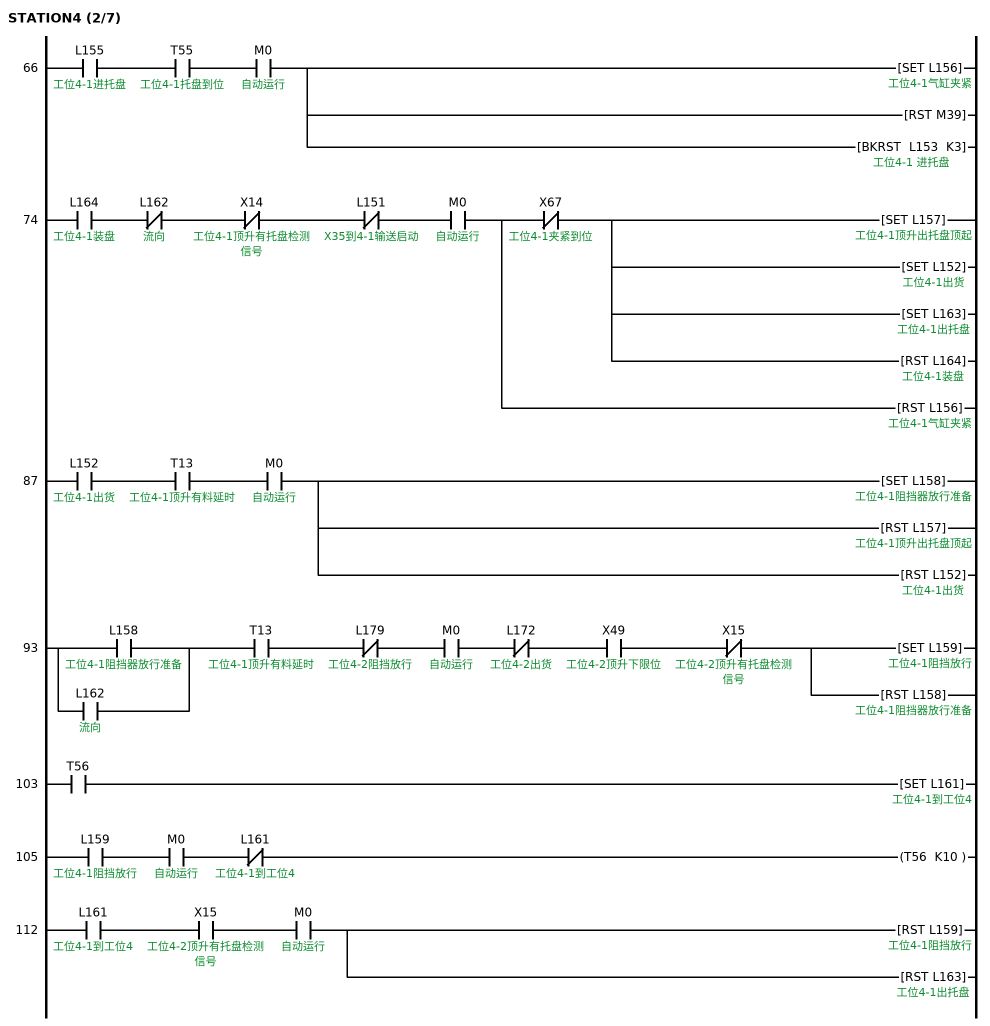
66    LD      L155  ; 工位4-1进托盘
      AND     T55  ; 工位4-1托盘到位
      AND     M0  ; 自动运行
      SET     L156  ; 工位4-1气缸夹紧
      RST     M39
      BKRST   L153 K3
74    LD      L164  ; 工位4-1装盘
      ANI     L162  ; 流向
      ANI     X14  ; 工位4-1顶升有托盘检测信号
      ANI     L151  ; X35到4-1输送启动
      AND     M0  ; 自动运行
      MPS
      ANI     X67  ; 工位4-1夹紧到位
      SET     L157  ; 工位4-1顶升出托盘顶起
      SET     L152  ; 工位4-1出货
      SET     L163  ; 工位4-1出托盘
      RST     L164  ; 工位4-1装盘
      MPP
      RST     L156  ; 工位4-1气缸夹紧
87    LD      L152  ; 工位4-1出货
      AND     T13  ; 工位4-1顶升有料延时
      AND     M0  ; 自动运行
      SET     L158  ; 工位4-1阻挡器放行准备
      RST     L157  ; 工位4-1顶升出托盘顶起
      RST     L152  ; 工位4-1出货
93    LD      L158  ; 工位4-1阻挡器放行准备
      OR      L162  ; 流向
      AND     T13  ; 工位4-1顶升有料延时
      ANI     L179  ; 工位4-2阻挡放行
      AND     M0  ; 自动运行
      ANI     L172  ; 工位4-2出货
      AND     X49  ; 工位4-2顶升下限位
      ANI     X15  ; 工位4-2顶升有托盘检测信号
      SET     L159  ; 工位4-1阻挡放行
      RST     L158  ; 工位4-1阻挡器放行准备
103   LD      T56
      SET     L161  ; 工位4-1到工位4
105   LD      L159  ; 工位4-1阻挡放行
      AND     M0  ; 自动运行
      ANI     L161  ; 工位4-1到工位4
      OUT     T56 K10
112   LD      L161  ; 工位4-1到工位4
      AND     X15  ; 工位4-2顶升有托盘检测信号
      AND     M0  ; 自动运行
      RST     L159  ; 工位4-1阻挡放行
      RST     L163  ; 工位4-1出托盘
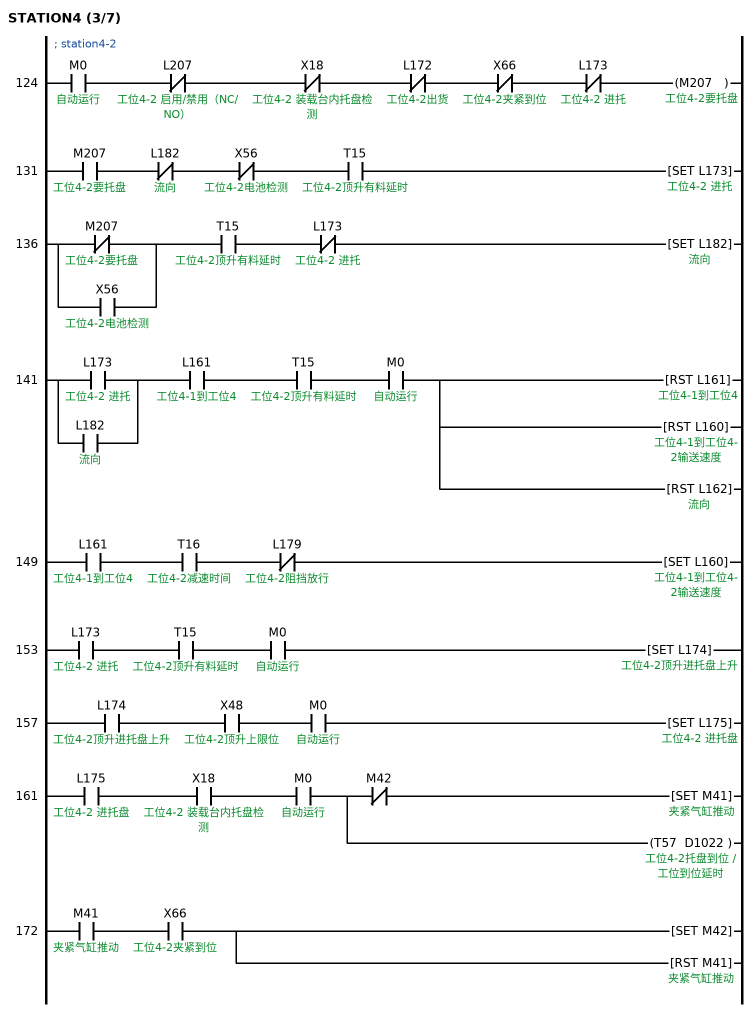
; station4-2
124   LD      M0  ; 自动运行
      ANI     L207  ; 工位4-2 启用/禁用（NC/NO）
      ANI     X18  ; 工位4-2 装载台内托盘检测
      ANI     L172  ; 工位4-2出货
      ANI     X66  ; 工位4-2夹紧到位
      ANI     L173  ; 工位4-2 进托
      OUT     M207  ; 工位4-2要托盘
131   LD      M207  ; 工位4-2要托盘
      ANI     L182  ; 流向
      ANI     X56  ; 工位4-2电池检测
      AND     T15  ; 工位4-2顶升有料延时
      SET     L173  ; 工位4-2 进托
136   LDI     M207  ; 工位4-2要托盘
      OR      X56  ; 工位4-2电池检测
      AND     T15  ; 工位4-2顶升有料延时
      ANI     L173  ; 工位4-2 进托
      SET     L182  ; 流向
141   LD      L173  ; 工位4-2 进托
      OR      L182  ; 流向
      AND     L161  ; 工位4-1到工位4
      AND     T15  ; 工位4-2顶升有料延时
      AND     M0  ; 自动运行
      RST     L161  ; 工位4-1到工位4
      RST     L160  ; 工位4-1到工位4-2输送速度
      RST     L162  ; 流向
149   LD      L161  ; 工位4-1到工位4
      AND     T16  ; 工位4-2减速时间
      ANI     L179  ; 工位4-2阻挡放行
      SET     L160  ; 工位4-1到工位4-2输送速度
153   LD      L173  ; 工位4-2 进托
      AND     T15  ; 工位4-2顶升有料延时
      AND     M0  ; 自动运行
      SET     L174  ; 工位4-2顶升进托盘上升
157   LD      L174  ; 工位4-2顶升进托盘上升
      AND     X48  ; 工位4-2顶升上限位
      AND     M0  ; 自动运行
      SET     L175  ; 工位4-2 进托盘
161   LD      L175  ; 工位4-2 进托盘
      AND     X18  ; 工位4-2 装载台内托盘检测
      AND     M0  ; 自动运行
      MPS
      ANI     M42
      SET     M41  ; 夹紧气缸推动
      MPP
      OUT     T57 D1022  ; 工位4-2托盘到位 / 工位到位延时
172   LD      M41  ; 夹紧气缸推动
      AND     X66  ; 工位4-2夹紧到位
      SET     M42
      RST     M41  ; 夹紧气缸推动
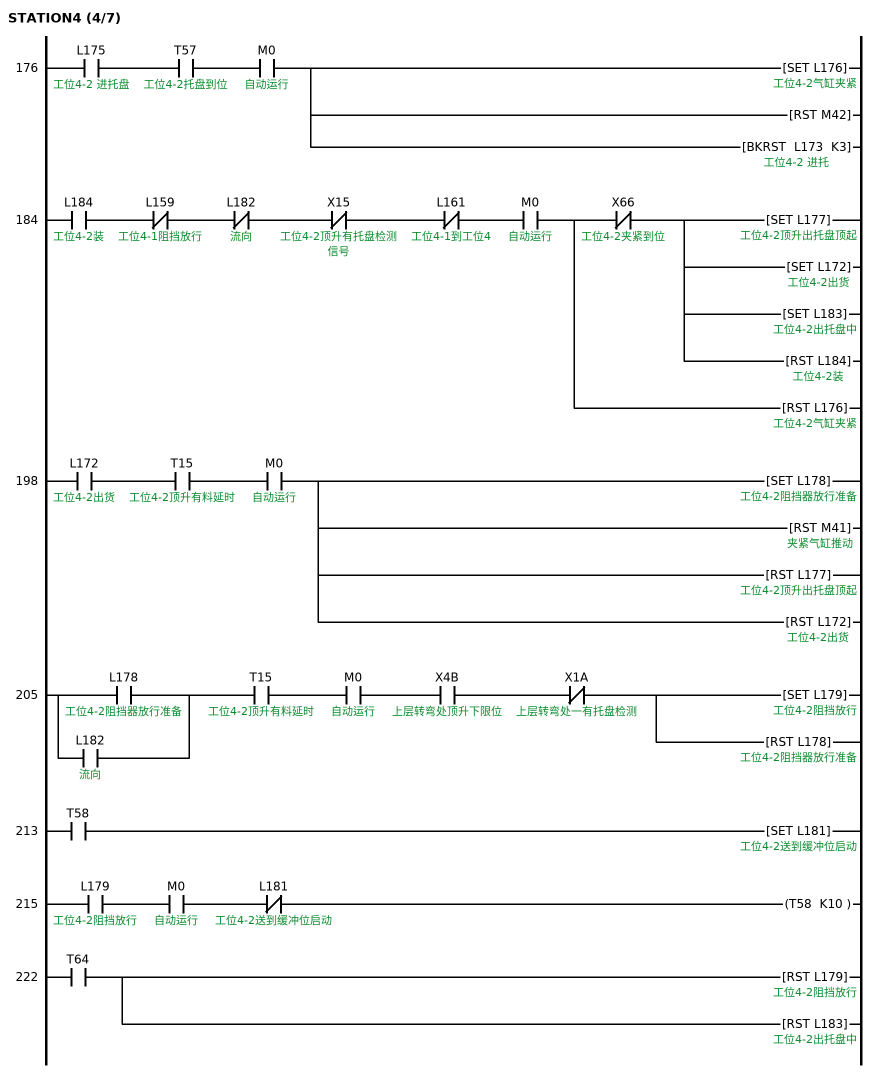
176   LD      L175  ; 工位4-2 进托盘
      AND     T57  ; 工位4-2托盘到位
      AND     M0  ; 自动运行
      SET     L176  ; 工位4-2气缸夹紧
      RST     M42
      BKRST   L173 K3
184   LD      L184  ; 工位4-2装
      ANI     L159  ; 工位4-1阻挡放行
      ANI     L182  ; 流向
      ANI     X15  ; 工位4-2顶升有托盘检测信号
      ANI     L161  ; 工位4-1到工位4
      AND     M0  ; 自动运行
      MPS
      ANI     X66  ; 工位4-2夹紧到位
      SET     L177  ; 工位4-2顶升出托盘顶起
      SET     L172  ; 工位4-2出货
      SET     L183  ; 工位4-2出托盘中
      RST     L184  ; 工位4-2装
      MPP
      RST     L176  ; 工位4-2气缸夹紧
198   LD      L172  ; 工位4-2出货
      AND     T15  ; 工位4-2顶升有料延时
      AND     M0  ; 自动运行
      SET     L178  ; 工位4-2阻挡器放行准备
      RST     M41  ; 夹紧气缸推动
      RST     L177  ; 工位4-2顶升出托盘顶起
      RST     L172  ; 工位4-2出货
205   LD      L178  ; 工位4-2阻挡器放行准备
      OR      L182  ; 流向
      AND     T15  ; 工位4-2顶升有料延时
      AND     M0  ; 自动运行
      AND     X4B  ; 上层转弯处顶升下限位
      ANI     X1A  ; 上层转弯处一有托盘检测
      SET     L179  ; 工位4-2阻挡放行
      RST     L178  ; 工位4-2阻挡器放行准备
213   LD      T58
      SET     L181  ; 工位4-2送到缓冲位启动
215   LD      L179  ; 工位4-2阻挡放行
      AND     M0  ; 自动运行
      ANI     L181  ; 工位4-2送到缓冲位启动
      OUT     T58 K10
222   LD      T64
      RST     L179  ; 工位4-2阻挡放行
      RST     L183  ; 工位4-2出托盘中
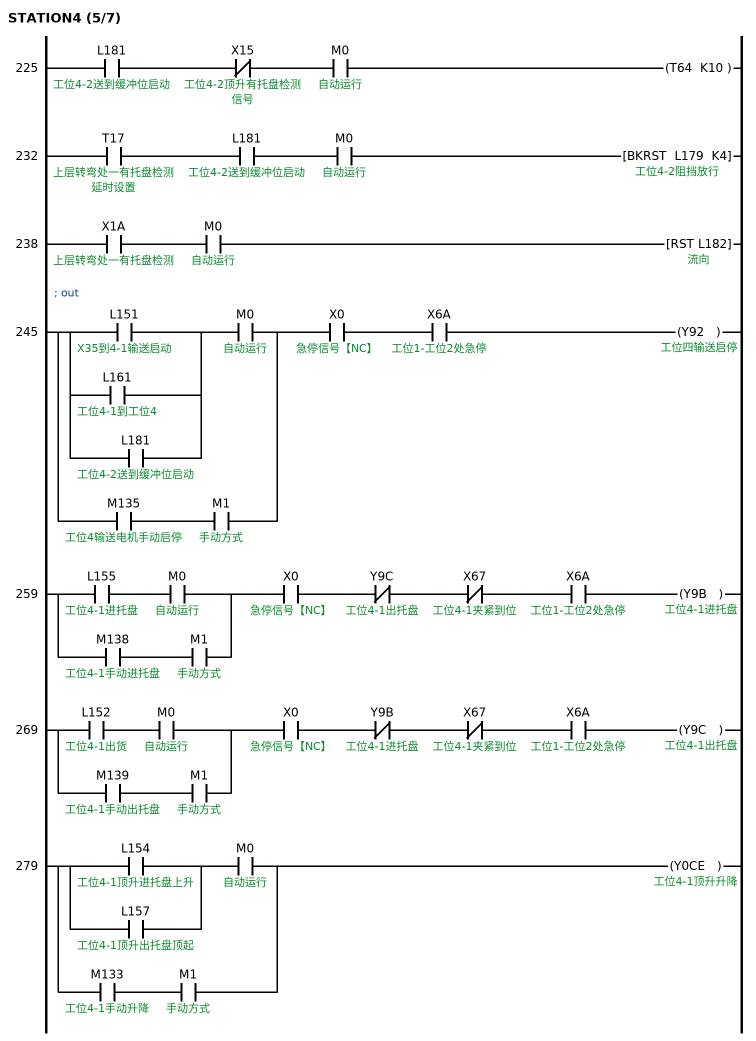
225   LD      L181  ; 工位4-2送到缓冲位启动
      ANI     X15  ; 工位4-2顶升有托盘检测信号
      AND     M0  ; 自动运行
      OUT     T64 K10
232   LD      T17  ; 上层转弯处一有托盘检测延时设置
      AND     L181  ; 工位4-2送到缓冲位启动
      AND     M0  ; 自动运行
      BKRST   L179 K4
238   LD      X1A  ; 上层转弯处一有托盘检测
      AND     M0  ; 自动运行
      RST     L182  ; 流向
; out
245   LD      L151  ; X35到4-1输送启动
      OR      L161  ; 工位4-1到工位4
      OR      L181  ; 工位4-2送到缓冲位启动
      AND     M0  ; 自动运行
      LD      M135  ; 工位4输送电机手动启停
      AND     M1  ; 手动方式
      ORB
      AND     X0  ; 急停信号【NC】
      AND     X6A  ; 工位1-工位2处急停
      OUT     Y92  ; 工位四输送启停
        [note] 4-1
259   LD      L155  ; 工位4-1进托盘
      AND     M0  ; 自动运行
      LD      M138  ; 工位4-1手动进托盘
      AND     M1  ; 手动方式
      ORB
      AND     X0  ; 急停信号【NC】
      ANI     Y9C  ; 工位4-1出托盘
      ANI     X67  ; 工位4-1夹紧到位
      AND     X6A  ; 工位1-工位2处急停
      OUT     Y9B  ; 工位4-1进托盘
269   LD      L152  ; 工位4-1出货
      AND     M0  ; 自动运行
      LD      M139  ; 工位4-1手动出托盘
      AND     M1  ; 手动方式
      ORB
      AND     X0  ; 急停信号【NC】
      ANI     Y9B  ; 工位4-1进托盘
      ANI     X67  ; 工位4-1夹紧到位
      AND     X6A  ; 工位1-工位2处急停
      OUT     Y9C  ; 工位4-1出托盘
279   LD      L154  ; 工位4-1顶升进托盘上升
      OR      L157  ; 工位4-1顶升出托盘顶起
      AND     M0  ; 自动运行
      LD      M133  ; 工位4-1手动升降
      AND     M1  ; 手动方式
      ORB
      OUT     Y0CE  ; 工位4-1顶升升降
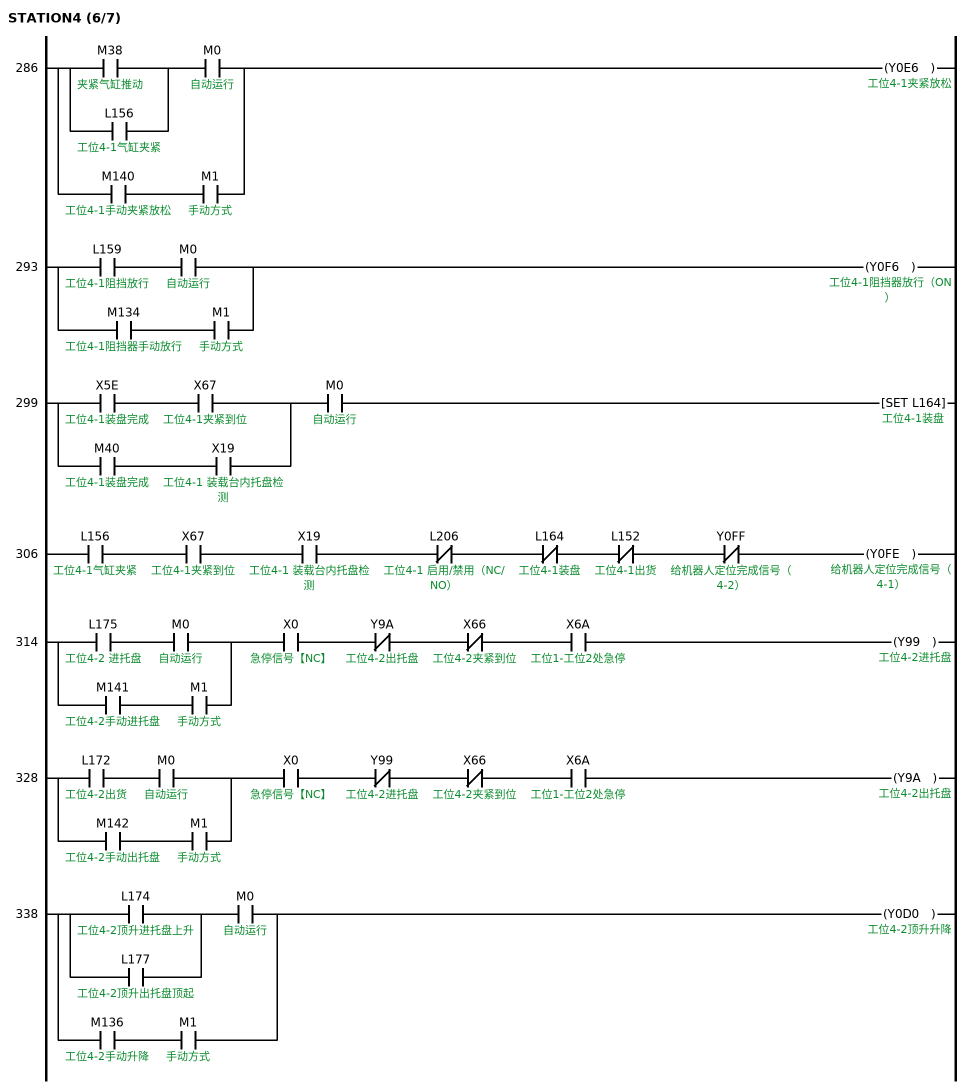
286   LD      M38  ; 夹紧气缸推动
      OR      L156  ; 工位4-1气缸夹紧
      AND     M0  ; 自动运行
      LD      M140  ; 工位4-1手动夹紧放松
      AND     M1  ; 手动方式
      ORB
      OUT     Y0E6  ; 工位4-1夹紧放松
293   LD      L159  ; 工位4-1阻挡放行
      AND     M0  ; 自动运行
      LD      M134  ; 工位4-1阻挡器手动放行
      AND     M1  ; 手动方式
      ORB
      OUT     Y0F6  ; 工位4-1阻挡器放行（ON）
299   LD      X5E  ; 工位4-1装盘完成
      AND     X67  ; 工位4-1夹紧到位
      LD      M40  ; 工位4-1装盘完成
      AND     X19  ; 工位4-1 装载台内托盘检测
      ORB
      AND     M0  ; 自动运行
      SET     L164  ; 工位4-1装盘
306   LD      L156  ; 工位4-1气缸夹紧
      AND     X67  ; 工位4-1夹紧到位
      AND     X19  ; 工位4-1 装载台内托盘检测
      ANI     L206  ; 工位4-1 启用/禁用（NC/NO）
      ANI     L164  ; 工位4-1装盘
      ANI     L152  ; 工位4-1出货
      ANI     Y0FF  ; 给机器人定位完成信号（4-2）
      OUT     Y0FE  ; 给机器人定位完成信号（4-1）
314   LD      L175  ; 工位4-2 进托盘
      AND     M0  ; 自动运行
      LD      M141  ; 工位4-2手动进托盘
      AND     M1  ; 手动方式
      ORB
      AND     X0  ; 急停信号【NC】
      ANI     Y9A  ; 工位4-2出托盘
      ANI     X66  ; 工位4-2夹紧到位
      AND     X6A  ; 工位1-工位2处急停
      OUT     Y99  ; 工位4-2进托盘
        [note] 4-2
328   LD      L172  ; 工位4-2出货
      AND     M0  ; 自动运行
      LD      M142  ; 工位4-2手动出托盘
      AND     M1  ; 手动方式
      ORB
      AND     X0  ; 急停信号【NC】
      ANI     Y99  ; 工位4-2进托盘
      ANI     X66  ; 工位4-2夹紧到位
      AND     X6A  ; 工位1-工位2处急停
      OUT     Y9A  ; 工位4-2出托盘
338   LD      L174  ; 工位4-2顶升进托盘上升
      OR      L177  ; 工位4-2顶升出托盘顶起
      AND     M0  ; 自动运行
      LD      M136  ; 工位4-2手动升降
      AND     M1  ; 手动方式
      ORB
      OUT     Y0D0  ; 工位4-2顶升升降
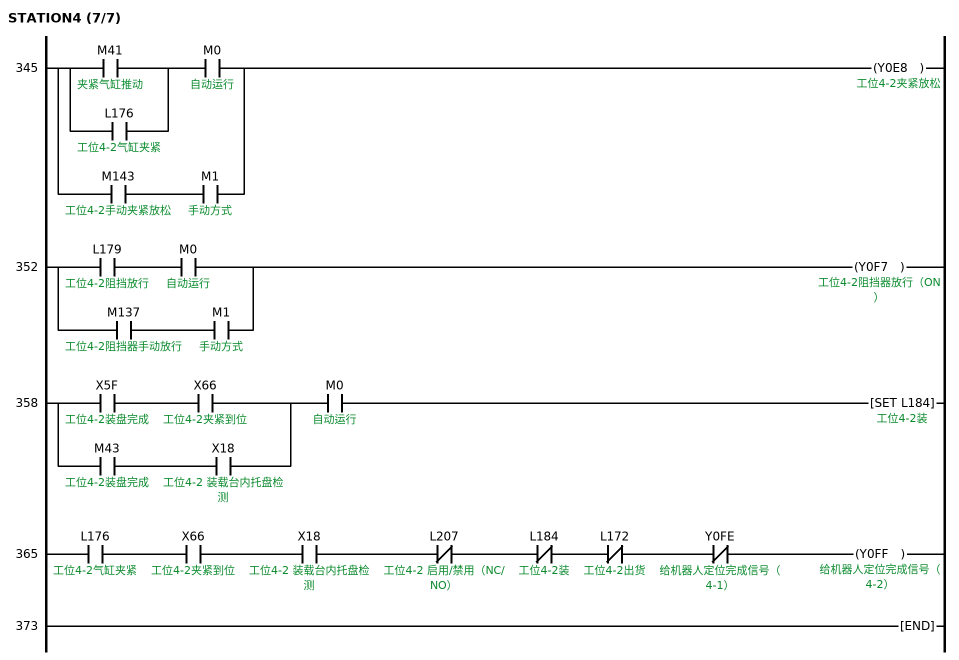
345   LD      M41  ; 夹紧气缸推动
      OR      L176  ; 工位4-2气缸夹紧
      AND     M0  ; 自动运行
      LD      M143  ; 工位4-2手动夹紧放松
      AND     M1  ; 手动方式
      ORB
      OUT     Y0E8  ; 工位4-2夹紧放松
352   LD      L179  ; 工位4-2阻挡放行
      AND     M0  ; 自动运行
      LD      M137  ; 工位4-2阻挡器手动放行
      AND     M1  ; 手动方式
      ORB
      OUT     Y0F7  ; 工位4-2阻挡器放行（ON）
358   LD      X5F  ; 工位4-2装盘完成
      AND     X66  ; 工位4-2夹紧到位
      LD      M43  ; 工位4-2装盘完成
      AND     X18  ; 工位4-2 装载台内托盘检测
      ORB
      AND     M0  ; 自动运行
      SET     L184  ; 工位4-2装
365   LD      L176  ; 工位4-2气缸夹紧
      AND     X66  ; 工位4-2夹紧到位
      AND     X18  ; 工位4-2 装载台内托盘检测
      ANI     L207  ; 工位4-2 启用/禁用（NC/NO）
      ANI     L184  ; 工位4-2装
      ANI     L172  ; 工位4-2出货
      ANI     Y0FE  ; 给机器人定位完成信号（4-1）
      OUT     Y0FF  ; 给机器人定位完成信号（4-2）
373   END
END_PROGRAM

PROGRAM TCP
VAR
  m_tonReconnect : TON;  (* 自动重连 *)
  m_xReconnect : BOOL;
  m_tReconnectCurrentTime : TIME;
  m_tonAutoClose : TON;  (* 自动关闭 *)
  m_xAutoClose : BOOL;
  m_tAutoCloseCurrentTime : TIME;
  m_ton1ReceiveHeartbeat : TON;  (* 心跳检查 *)
  m_t1RecHeartbeatCurrentTime : TIME;
  m_xOpenSuccess : BOOL;  (* 打开成功 *)
  m_xSendSuccess : BOOL;  (* 发送成功 *)
  m_xReceiveSuccess : BOOL;  (* 接收成功 *)
  m_iOpenCtrl : INT;  (* 打开指令控制字 *)
  m_iSendCtrl : INT;  (* 发送指令控制字 *)
  m_iReceivectrl : INT;  (* 接收指令控制字 *)
  m_iClosectrl : INT;  (* 关闭指令控制字 *)
  m_xCloseSuccess : BOOL;  (* 关闭成功 *)
END_VAR
D200:=4;
D201:=H54;(*16进制的54就是T，扫码枪设定的扫码触发条件*)
m_tonReconnect(IN:= NOT SD1282.0 AND NOT SD1284.0  ,PT:=T#5s  ,Q:=m_xReconnect ,ET:=m_tReconnectCurrentTime);
SP_SOCOPEN(m_xReconnect  AND SD1288.A , "U0", K1 , D100, M900);
SP_SOCSND( LDP(TRUE,g_xScan) AND SD1282.0 , "U0" , K1 , D110, D200, M910);
SP_SOCRCV( SD1282.0 AND SD1286.0 AND NOT M920, "U0" , K1, D120, g_iBatteryInformation[0],M920);
m_tonAutoClose(IN:= SD1284.0 AND NOT SD1282.0 ,PT:=T#5s,Q:=m_xAutoClose ,ET:= m_tAutoCloseCurrentTime );
SP_SOCCLOSE( LDF(TRUE,SD1282.0) OR m_xAutoClose  , "U0" , K1, D130, M930);
END_PROGRAM

PROGRAM TP-LINE
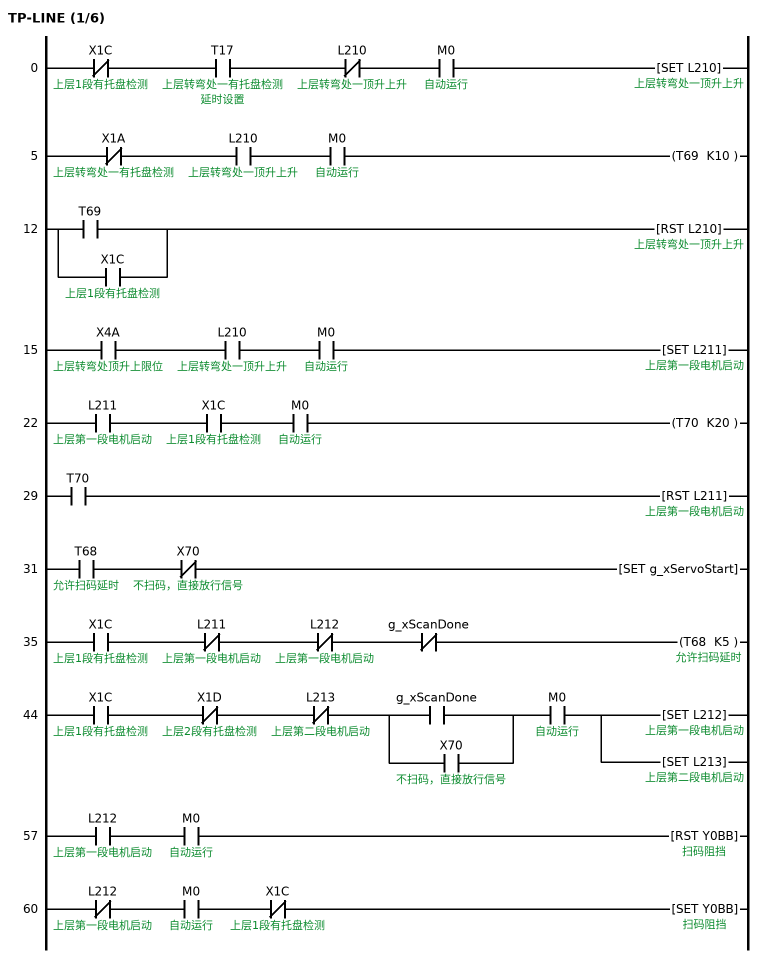
0     LDI     X1C  ; 上层1段有托盘检测
      AND     T17  ; 上层转弯处一有托盘检测延时设置
      ANI     L210  ; 上层转弯处一顶升上升
      AND     M0  ; 自动运行
      SET     L210  ; 上层转弯处一顶升上升
5     LDI     X1A  ; 上层转弯处一有托盘检测
      AND     L210  ; 上层转弯处一顶升上升
      AND     M0  ; 自动运行
      OUT     T69 K10
12    LD      T69
      OR      X1C  ; 上层1段有托盘检测
      RST     L210  ; 上层转弯处一顶升上升
15    LD      X4A  ; 上层转弯处顶升上限位
      AND     L210  ; 上层转弯处一顶升上升
      AND     M0  ; 自动运行
      SET     L211  ; 上层第一段电机启动
        [note] 1
22    LD      L211  ; 上层第一段电机启动
      AND     X1C  ; 上层1段有托盘检测
      AND     M0  ; 自动运行
      OUT     T70 K20
29    LD      T70
      RST     L211  ; 上层第一段电机启动
31    LD      T68  ; 允许扫码延时
      ANI     X70  ; 不扫码，直接放行信号
      SET     g_xServoStart
35    LD      X1C  ; 上层1段有托盘检测
      ANI     L211  ; 上层第一段电机启动
      ANI     L212  ; 上层第一段电机启动
      ANI     g_xScanDone
      OUT     T68 K5  ; 允许扫码延时
44    LD      X1C  ; 上层1段有托盘检测
      ANI     X1D  ; 上层2段有托盘检测
      ANI     L213  ; 上层第二段电机启动
      LD      g_xScanDone
      OR      X70  ; 不扫码，直接放行信号
      ANB
      AND     M0  ; 自动运行
      SET     L212  ; 上层第一段电机启动
        [note] 2
      SET     L213  ; 上层第二段电机启动
57    LD      L212  ; 上层第一段电机启动
      AND     M0  ; 自动运行
      RST     Y0BB  ; 扫码阻挡
60    LDI     L212  ; 上层第一段电机启动
      AND     M0  ; 自动运行
      ANI     X1C  ; 上层1段有托盘检测
      SET     Y0BB  ; 扫码阻挡
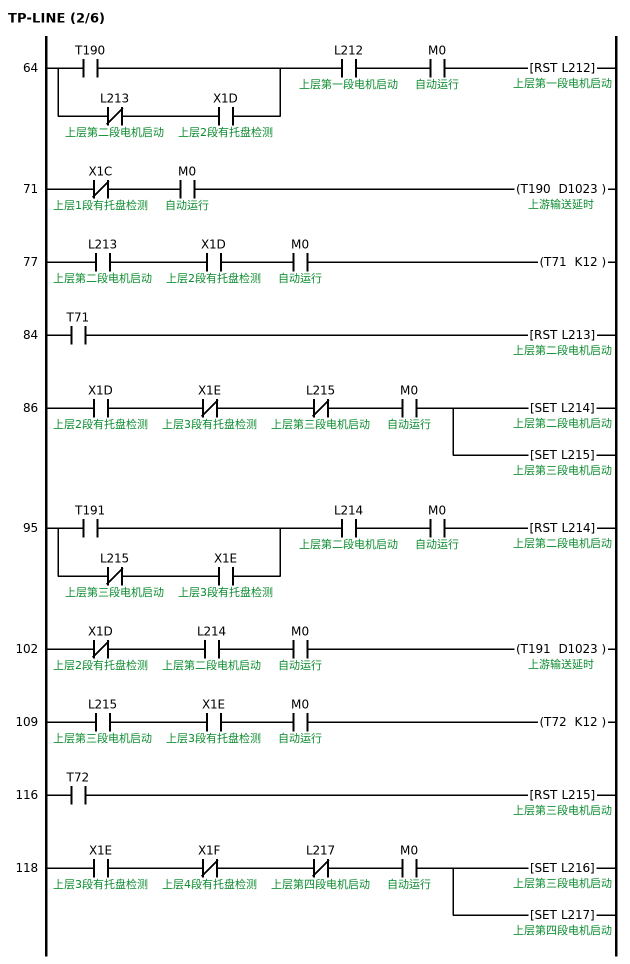
64    LD      T190
      LDI     L213  ; 上层第二段电机启动
      AND     X1D  ; 上层2段有托盘检测
      ORB
      AND     L212  ; 上层第一段电机启动
      AND     M0  ; 自动运行
      RST     L212  ; 上层第一段电机启动
71    LDI     X1C  ; 上层1段有托盘检测
      AND     M0  ; 自动运行
      OUT     T190 D1023  ; 上游输送延时
77    LD      L213  ; 上层第二段电机启动
      AND     X1D  ; 上层2段有托盘检测
      AND     M0  ; 自动运行
      OUT     T71 K12
84    LD      T71
      RST     L213  ; 上层第二段电机启动
86    LD      X1D  ; 上层2段有托盘检测
      ANI     X1E  ; 上层3段有托盘检测
      ANI     L215  ; 上层第三段电机启动
      AND     M0  ; 自动运行
      SET     L214  ; 上层第二段电机启动
        [note] 3
      SET     L215  ; 上层第三段电机启动
95    LD      T191
      LDI     L215  ; 上层第三段电机启动
      AND     X1E  ; 上层3段有托盘检测
      ORB
      AND     L214  ; 上层第二段电机启动
      AND     M0  ; 自动运行
      RST     L214  ; 上层第二段电机启动
102   LDI     X1D  ; 上层2段有托盘检测
      AND     L214  ; 上层第二段电机启动
      AND     M0  ; 自动运行
      OUT     T191 D1023  ; 上游输送延时
109   LD      L215  ; 上层第三段电机启动
      AND     X1E  ; 上层3段有托盘检测
      AND     M0  ; 自动运行
      OUT     T72 K12
116   LD      T72
      RST     L215  ; 上层第三段电机启动
118   LD      X1E  ; 上层3段有托盘检测
      ANI     X1F  ; 上层4段有托盘检测
      ANI     L217  ; 上层第四段电机启动
      AND     M0  ; 自动运行
      SET     L216  ; 上层第三段电机启动
        [note] 4
      SET     L217  ; 上层第四段电机启动
